FUNCTION_BLOCK "GCS7_M_Mixer"	// FB 54
TITLE = Mixer: Motor with 2 Digital Input
//  
//COPYRIGHT:    (C) 1997  BUHLER AG, CH-9240 UZWIL,  SWITZERLAND
//
//PRODUCT:      GCS7
//
//TITLE:        FB 54 MACHINE-CONTROL:Mixer:Motor with 2 Digital Input
//
//-------------------------------------------------------------------------
//
//IDENT:        AUTHOR:             DEPT:                       DATE:
//
//FB54.4.0      A. Egli             CT3                         17-Jun-2002
//              New Release with one block 
//FB54.3.1      A. Egli             CT3                         20-Mar-2000
//              Reset after mix done if mixer is open 
//FB54.3.0      A. Egli             CT3                         11-Oct-1999
//              Local data reduced 
//FB54.2B       K. Tischer          MU664                       06-Mar-1999
//              CC FC2 not UC FC2
//FB54.2A       A. Egli             CT3                         04-Mai-1998
//              StFault = StCode 32
//FB54.1A       A.Egli              AEE61                       5-Jul-1997
//              1st Release in S7
//
//-------------------------------------------------------------------------
//
//PURPOSE:      MANUAL : see [LL.MIXxxMAN]
//
//RESTRICTIONS: S7
//              ACCU2: Pointer to dynamic datas of the machine
//              ACCU1: Pointer to parameter datas of the machine
//
//-------------------------------------------------------------------------
//
AUTHOR : EA
FAMILY : GCS7LL
NAME : Mixer
VERSION : 4.0
VAR
  Ma : UDT 20540;
  Mon1 : FB 14;	//Element
  Mon2 : FB 14;	//Element
  Motor : FB 12;	//Element
END_VAR
VAR_TEMP
  tmpFaultStop : BOOL ;
  tmpFaultSum : BOOL ;
  tmpLocal : BOOL ;
  tmpLenDyn : INT ;
END_VAR
BEGIN
NETWORK
TITLE =
      L     22;
      T     #tmpLenDyn;
NETWORK
TITLE = PC Control
//=== Test Object number =====================
      L     "SYS_DirectCtrlDB".PC.ObjectNo;	//PCControl.ObjectNo
      L     #Ma.Par.ParObjectNo;	//Input ObjectNo
      <>I;
      JC    aEnd;
//=== Test OType      ========================
      L     2054;	//Input object type
      L     "SYS_DirectCtrlDB".PC.ObjectType;	//PCControl.ObjectType
      <>I;
      JC    aEnd;
//=== Test Handshake =========================
      A     "SYS_DirectCtrlDB".PC.Hsk.FExamine;	// Handshake.FExamine
      JC    aExa;
      A     "SYS_DirectCtrlDB".PC.Hsk.FDefineCmd;	// Handshake.FDefineCmd
      JC    aCmd;
      A     "SYS_DirectCtrlDB".PC.Hsk.FDefinePara;	// Handshake.FDefinePara
      JC    aPar;
aIni: L     2;	// FcInit
      UC    "SYS_DirectCtrl";
      JU    aEnd;
// Write parameter 
aPar: LAR1  P#DBX 58.0;
      L     P#6.0;
      +AR1;
      L     DBW [AR1,P#4.0];
      T     #Ma.Par.ParAfterMixTime;
// Write new commands from PC to Interface of group 
aCmd: A     "SYS_DirectCtrlDB".PC.Cmd1[8];	//Cmd1[8]=CmdOff
      S     #Ma.CmdOff;
      A     "SYS_DirectCtrlDB".PC.Cmd1[9];	//Cmd1[9]=CmdOn
      S     #Ma.CmdOn;
      A     "SYS_DirectCtrlDB".PC.Cmd1[10];	//Cmd1[10]=CmdNext
      S     #Ma.CmdNext;
      A     "SYS_DirectCtrlDB".PC.Cmd1[11];	//Cmd1[11]=CmdFaultReset
      S     #Ma.CmdFaultReset;
      A     "SYS_DirectCtrlDB".PC.Cmd1[13];	//Cmd1[13]=CmdManualOn
      S     #Ma.InManual;
      A     "SYS_DirectCtrlDB".PC.Cmd2[13];	//Cmd2[13]=CmdManualOff
      R     #Ma.InManual;
      A     "SYS_DirectCtrlDB".PC.Cmd1[6];	//Cmd1[14]=SlowOn
      S     #Motor.InOutManSlow;
      A     "SYS_DirectCtrlDB".PC.Cmd2[6];	//Cmd2[14]=SlowOff
      R     #Motor.InOutManSlow;
//Define Value
      AN    "SYS_DirectCtrlDB".PC.Hsk.FDefineValue;	// PC.Hsk.FDefineValue
      ON    #Ma.InManual;
      JC    aIni;
      LAR1  P#DBX 58.0;
      L     DBW [AR1,P#6.0];
      T     #Ma.InPreMixTime;
      L     DBW [AR1,P#8.0];
      T     #Ma.InMainMixTime;
      JU    aIni;
aExa: TAR2;	// Address Dynamic datas
      T     "SYS_DirectCtrlDB".GC.InDynAddr;	// -->PCControl.GC.InDynAddr
      L     #tmpLenDyn;	// Length Dynamic data
      T     "SYS_DirectCtrlDB".GC.InDynLen;	// -->PCControl.GC.InDynLen
      L     0;
      T     "SYS_DirectCtrlDB".GC.InParaAddr;	// -->PCControl.GC.InParaAddr
      T     "SYS_DirectCtrlDB".GC.InParaLen;	// -->PCControl.GC.InParaLen
      L     1;	// Code FcExamine
      UC    "SYS_DirectCtrl";
      L     10;	//Revision
      T     "SYS_DirectCtrlDB".GC.Revision;
aEnd: NOP   0;
NETWORK
TITLE = Interlocking
//===Global Group Orders===
      A     "GCS7_Gr_OutManualOn";	//Gr.OutManualOn
      S     #Ma.InManual;
      A     "GCS7_Gr_OutManualOff";	//Gr.OutManualOff
      R     #Ma.InManual;
      A     #Ma.InManual;
      S     "GCS7_Gr_InManual";	//Gr.InManual
      A     #Ma.InLocal;
      AN    #Ma.InManual;
      =     #tmpLocal;
//---Emptied
      A     #Ma.OutMainMixDone;
      A     #Ma.InOpen;
      S     #Ma.OutEmptied;
      AN    #Ma.OutMainMixDone;
      R     #Ma.OutEmptied;
//----New batch
      AN    #Ma.InRunPreMix;
      AN    #Ma.InRunMainMix;
      O     #Ma.CmdNewBatch;
      R     #Ma.OutEmptied;
      R     #Ma.OutPreMixIsOn;
      R     #Ma.OutPreMixDone;
//--- Fault----
      A     #Mon1.StFault;
      O     #Mon2.StFault;
      O     #Motor.StFault;
      =     #tmpFaultSum;
      =     #tmpFaultStop;
//--- Motor----
      AN    #Ma.OutAfterMixDone;
      O     #Ma.OutEmptied;
      O     #Ma.InManual;
      A     #Ma.InEnable;
      AN    #tmpFaultStop;
      A(;
      A     #Mon2.InpTrue;
      O     #Ma.Par.ParMon2IsLS;
      ON    #Ma.Par.ParWithMon2;
      );
      A(;
      A     #Mon1.InpTrue;
      ON    #Ma.Par.ParWithMon1;
      );
      AN    #Ma.CmdOff;
      =     #Motor.InEnableFwd;
      AN    #Ma.OutMainMixDone;
      O     #Ma.OutEmptied;
      A     #Ma.CmdNext;
      AN    #Ma.InManual;
      O;
      A     #Ma.InManual;
      A     #Ma.CmdOn;
      S     #Motor.CmdNext;
      A     #Ma.InSeqStop;
      AN    #Ma.InManual;
      =     #Motor.InSeqStop;
//--- Local mode --
      A     #tmpLocal;
      =     #Motor.InLocal;
      A     #Motor.StStopped;
      A     #tmpLocal;
      =     #Mon1.InLocal;
      =     #Mon2.InLocal;
//--- Monitoring
      SET;
      =     #Mon1.InMonTrue;
      A     #Motor.StStartedFwd;
      O     #Motor.StStartedRev;
      O     #Ma.Par.ParMon2IsLS;
      =     #Mon2.InMonTrue;
//--- Fault Reset -------------
      A     #Ma.CmdFaultReset;
      S     #Motor.CmdFaultReset;
      S     #Mon1.CmdFaultReset;
      S     #Mon2.CmdFaultReset;
NETWORK
TITLE = Mixing time
      L     0;
      L     #Ma.OutMixTime;
      >=I;
      JC    mix;
      AN    "GCS7_Gr_OutTick1s";	//Gr.OutTick1s
      ON    #Motor.StStartedFwd;
      JC    mix;
      +     -1;
      T     #Ma.OutMixTime;
//Pre mixing time 
mix:  AN    #Ma.InRunPreMix;
      AN    #Ma.InRunMainMix;
      R     #Ma.OutPreMixIsOn;
      R     #Ma.OutPreMixDone;
      JC    m2;
      A     #Ma.OutPreMixDone;
      JC    m2;
      A     #Ma.OutPreMixIsOn;
      JC    m12;
      S     #Ma.OutPreMixIsOn;
      L     #Ma.InPreMixTime;
      T     #Ma.OutMixTime;
m12:  L     #Ma.OutMixTime;
      L     0;
      <=I;
      R     #Ma.OutPreMixIsOn;
      S     #Ma.OutPreMixDone;
//Main mixing time 
m2:   AN    #Ma.InRunMainMix;
      ON    #Ma.OutPreMixDone;
      R     #Ma.OutMainMixIsOn;
      R     #Ma.OutMainMixDone;
      JC    m3;
      A     #Ma.OutMainMixDone;
      JC    m3;
      A     #Ma.OutMainMixIsOn;
      JC    m22;
      S     #Ma.OutMainMixIsOn;
      L     #Ma.InMainMixTime;
      T     #Ma.OutMixTime;
m22:  L     #Ma.OutMixTime;
      L     0;
      <=I;
      R     #Ma.OutMainMixIsOn;
      S     #Ma.OutMainMixDone;
//After mixing time 
m3:   AN    #Ma.OutMainMixDone;
      O     #Ma.InOpen;
      O     #Ma.OutEmptied;
      R     #Ma.OutAfterMixIsOn;
      R     #Ma.OutAfterMixDone;
      JC    m4;
      A     #Ma.OutAfterMixDone;
      JC    m4;
      A     #Ma.OutAfterMixIsOn;
      JC    m32;
      S     #Ma.OutAfterMixIsOn;
      L     #Ma.Par.ParAfterMixTime;
      T     #Ma.OutMixTime;
m32:  L     #Ma.OutMixTime;
      L     0;
      <=I;
      R     #Ma.OutAfterMixIsOn;
      S     #Ma.OutAfterMixDone;
NETWORK
TITLE = Call Digital Input: Monitor B1
m4:   AN    #Ma.Par.ParWithMon1;
      JC    m5;
      CALL  #Mon1;
NETWORK
TITLE = Call Digital Input: Monitor B2
m5:   AN    #Ma.Par.ParWithMon2;
      JC    Moto;
      CALL  #Mon2;
NETWORK
TITLE = Call Motor
Moto: CALL  #Motor;
NETWORK
TITLE = Jump to actual state
      A     #Ma.StStopped;
      JC    S0;	// ===> State
      A     #Ma.StStarted;
      JC    S2;	// ===> State
      A     #Ma.StStarting;
      JC    S1;	// ===> State
      A     #Ma.StStopping;
      JC    S3;	// ===> State
      A     #Ma.StFault;
      JC    S4;	// ===> State
NETWORK
TITLE = Stopped
xxS0: S     #Ma.StStopped;
S0:   A     #tmpFaultSum;
      R     #Ma.StStopped;
      JC    xxS4;	//--> StFault
      AN    #Motor.StStopped;
      R     #Ma.StStopped;
      JC    xxS1;	//--> StStarting
      JU    OUT;
NETWORK
TITLE = Starting
xxS1: S     #Ma.StStarting;
S1:   A     #tmpFaultSum;
      R     #Ma.StStarting;
      JC    xxS4;	//--> StFault
// Condition for StStopping
      A     #Motor.StStopped;
      O     #Motor.StStopping;
      R     #Ma.StStarting;
      JC    xxS3;	//--> StStopping
      AN    #Mon1.StTrue;
      A     #Ma.Par.ParWithMon1;
      O;
      AN    #Mon2.StTrue;
      A     #Ma.Par.ParWithMon2;
      JC    S2En;
// Condition for StStartedFwd
      A     #Motor.StStartedFwd;
      R     #Ma.StStarting;
      JC    xxS2;	//--> StStartedFwd
S2En: JU    OUT;
NETWORK
TITLE = StartedFwd
xxS2: S     #Ma.StStarted;
S2:   A     #tmpFaultSum;
      R     #Ma.StStarted;
      JC    xxS4;	//--> StFault
// Condition for StStopping
      AN    #Motor.StStartedFwd;
      R     #Ma.StStarted;
      JC    xxS3;	//--> StStopping
      JU    OUT;
NETWORK
TITLE = Stopping
xxS3: S     #Ma.StStopping;
S3:   A     #tmpFaultSum;
      R     #Ma.StStopping;
      JC    xxS4;	//--> StFault
// Condition for StStopped
      A     #Motor.StStopped;
      R     #Ma.StStopping;
      JC    xxS0;	//--> StStopped
// Condition for StStarting
      AN    #Motor.StStopping;
      R     #Ma.StStopping;
      JC    xxS1;	//--> StStarting
      JU    OUT;
NETWORK
TITLE = Fault
xxS4: S     #Ma.StFault;
S4:   AN    #tmpFaultSum;
      R     #Ma.StFault;
      JC    xxS3;	//--> StStopping
      JU    OUT;
NETWORK
TITLE = Global End
OUT:  CLR;	//---Clear all commands
      =     #Ma.CmdOn;
      =     #Ma.CmdOff;
      =     #Ma.CmdNext;
      =     #Ma.CmdFaultReset;
      =     #Ma.CmdNewBatch;
NETWORK
TITLE = State Code
// Same as motor
      L     32;	// StCode=Fault
      A     #Ma.StFault;
      JC    Code;
//Started
      AN    #Ma.StStarted;
      JC    C2;
      A     #Ma.OutPreMixIsOn;
      AN    #Ma.OutEmptied;
      L     4;	// StCode=Premix
      JC    Code;
      A     #Ma.OutMainMixIsOn;
      AN    #Ma.OutEmptied;
      L     5;	// StCode=MainMix
      JC    Code;
      A     #Ma.OutAfterMixIsOn;
      AN    #Ma.OutEmptied;
      L     6;	// StCode=AfterMix
      JC    Code;
      L     3;	// StCode=Started
      JU    Code;
//Stopped
C2:   AN    #Ma.StStopped;
      JC    C1;
      A     #Ma.OutMainMixDone;
      AN    #Ma.OutEmptied;
      L     8;	// StCode=Wait
      JC    Code;
      L     1;	// StCode=Stopped
      JU    Code;
//Starting
C1:   A     #Ma.StStarting;
      L     2;	// StCode=Starting
      JC    Code;
//Stopping
      L     7;	// StCode=Stopping
Code: L     #Ma.StCode;	// Old state code
      TAK;
      T     #Ma.StCode;	// Save state code
      <>I;
      L     3;
      CC    "SYS_CBitCtrl";	//Set change bit
END_FUNCTION_BLOCK

FUNCTION_BLOCK "GCS7_M_DFZK"	// FB 55
TITLE = DFZK vertical rotor mill
//  
//COPYRIGHT:    (C) 2000  BUHLER AG, CH-9240 UZWIL, SWITZERLAND
//
//PRODUCT:      GCS7
//
//TITLE:        FB55 Machine Control: DFZK vertical rotor mill
//
//-------------------------------------------------------------------------
//
//IDENT:        AUTHOR:             DEPT:                       DATE:
//
//FB55.2.3      A.Egli              CT3                         21.1.2005
//              For Screen change check input button
//FB55.2.2      A.Egli              FU53                        18.05.2004
//              Reset Manual mode when mill is not in automatic
//FB55.2.1      A.Egli              FU53                        15.03.2004
//              DFCM Freigabe koordinieren
//              Transition to StStopping if only one of both mill used
//              (Change [1.6] and [1.6a] from B.Thoma 
//FB55.2.0      A. Egli             CT3                         17-Jun-2002
//              New Release with one block 
//FB55.1.5      A.Egli              CT3                         14.09.2001
//              Condition B201LS.InMonTrue,B250LS.InMonTrue
//FB55.1.4      A.Egli              CT3                         14.09.2001
//              Unlock Cone in StNoPosition 
//FB55.1.3      B.Thoma             FU53                        21.01.2001
//              Monitoring Metal purifying if ma.ststarted 
//FB55.1.2      S. Kalberer         CT3                         21.11.2000
//              Avoid simultaneous brake event with global flag M 12.0
//FB55.1.1      S. Kalberer         CT3                         02.10.2000
//              Process of elements B201LS + 250LS (clam-gates) adapted
//FB55.1.0      S. Kalberer         CT3                         06.06.2000
//              1st Release in S7
//FB55.0.3      S. Kalberer         CT3                         26.05.2000
//              Cone open/close adapted
//FB55.0.2      S. Kalberer         CT3                         03.05.2000
//              Empty run without DFCM
//FB55.0.1      S. Kalberer         CT3                         26.04.2000
//              Segment gate parameter changed
//FB55.0.0      S. Kalberer         CT3                         20.04.2000
//              Software brake event and speed change
//
//-------------------------------------------------------------------------
//
//PURPOSE:      MANUAL : see [LL.VRMillENMAN]
//
//RESTRICTIONS: S7
//              ACCU2: Pointer to dynamic datas of the machine
//              ACCU1: Pointer to parameter datas of the machine
//
//-------------------------------------------------------------------------
//
AUTHOR : EA
FAMILY : GCS7LL
NAME : DFZKVRMi
VERSION : 2.3
VAR
  Ma : UDT 20550;
  M200 : FB 12;	//Element
  M300 : FB 12;	//Element
  M350 : FB 12;	//Element
  DFCMMill1 : FB 12;	//Element
  DFCMMill2 : FB 12;	//Element
  Y203V : FB 13;	//Element
  Y302V_Y305V : FB 13;	//Element
  Y352V_Y355V : FB 13;	//Element
  Y307V_Y309V : FB 13;	//Element
  Y357V_Y359V : FB 13;	//Element
  A316VI : FB 14;	//Element
  A366VI : FB 14;	//Element
  B205LS : FB 14;	//Element
  B206HL : FB 14;	//Element
  B201LS : FB 14;	//Element
  B250LS : FB 14;	//Element
  B300SM : FB 14;	//Element
  B350SM : FB 14;	//Element
  B310LS : FB 14;	//Element
  B360LS : FB 14;	//Element
  B317HL : FB 14;	//Element
  B367HL : FB 14;	//Element
  A209LC_AO1 : FB 17;	//Element
  A209LC_AO2 : FB 17;	//Element
  A209LC_AI1 : FB 19;	//Element
  A209LC_AI2 : FB 19;	//Element
  Y251V_52_53_54V : FB 20;	//Element
END_VAR
VAR_TEMP
  tmpFaultSum : BOOL ;	// Summary faults
  tmpFaultStopFeedingMill1 : BOOL ;	// Relevant faults to stop feeding mill 1
  tmpFaultStopFeedingMill2 : BOOL ;	// Relevant faults to stop feeding mill 2
  tmpFaultImmStopMill1 : BOOL ;	// Relevant faults to stop mill 1 immediately
  tmpFaultImmStopMill2 : BOOL ;	// Relevant faults to stop mill 2 immediately
  tmpFaultStopAfEmptyMill1 : BOOL ;	// Relevant faults to stop mill 2 after emptying time
  tmpFaultStopAfEmptyMill2 : BOOL ;	// Relevant faults to stop mill 1 after emptying time
  tmpEnableMill1 : BOOL ;
  tmpEnableMill2 : BOOL ;	//[1.2] ParMa.OutScreenChMill1 = tmpOutScreenChangeMill1 : BOOL; // Signal screen
  tmpSpeedChangeMill1 : BOOL ;	// Speed change requested mill 1
  tmpSpeedChangeMill2 : BOOL ;	// Speed change requested mill 1
  tmpTriggerFlag : BOOL ;
  tmpLenDyn : INT ;
END_VAR
BEGIN
NETWORK
TITLE =
      L     106;
      T     #tmpLenDyn;
NETWORK
TITLE = PC Control
//=== Test Object number =====================
      L     "SYS_DirectCtrlDB".PC.ObjectNo;	//PCControl.ObjectNo
      L     #Ma.Par.ParObjectNo;	//Input ObjectNo
      <>I;
      JC    aEnd;
//=== Test OType  ========================
      L     2055;	//Input object type
      L     "SYS_DirectCtrlDB".PC.ObjectType;	//PCControl.ObjectType
      <>I;
      JC    aEnd;
//=== Test Handshake =========================
      A     "SYS_DirectCtrlDB".PC.Hsk.FExamine;	// Handshake.FExamine
      JC    aExa;
      A     "SYS_DirectCtrlDB".PC.Hsk.FDefineCmd;	// Handshake.FDefineCmd
      JC    aCmd;
      A     "SYS_DirectCtrlDB".PC.Hsk.FDefinePara;	// Handshake.FDefinePara
      JC    pPar;
aIni: L     2;	// FcInit
      UC    "SYS_DirectCtrl";
      JU    aEnd;
// Write parameter 
pPar: LAR1  P#DBX 58.0;
      L     P#6.0;
      +AR1;
      L     DBW [AR1,P#4.0];
      L     "SYS_DirectCtrlDB".PC.Value[25];	//PCControl.PC.Value[25]
      T     #Ma.Par.ParEmptyRunMill1;
      L     "SYS_DirectCtrlDB".PC.Value[26];	//PCControl.PC.Value[26]
      T     #Ma.Par.ParEmptyRunMill2;
      L     "SYS_DirectCtrlDB".PC.Value[27];	//PCControl.PC.Value[27]
      T     #Ma.Par.ParEmptyTimeMill1;
      L     "SYS_DirectCtrlDB".PC.Value[28];	//PCControl.PC.Value[28]
      T     #Ma.Par.ParEmptyTimeMill2;
      L     "SYS_DirectCtrlDB".PC.Value[29];	//PCControl.PC.Value[29]
      T     #Ma.Par.ParBrakeTimeMill1;
      L     "SYS_DirectCtrlDB".PC.Value[30];	//PCControl.PC.Value[30]
      T     #Ma.Par.ParBrakeTimeMill2;
      L     "SYS_DirectCtrlDB".PC.Value[31];	//PCControl.PC.Value[31]
      T     #Ma.Par.ParSwitchChTime;
// Write new commands from PC to Interface of group 
aCmd: A     "SYS_DirectCtrlDB".PC.Cmd1[0];	//Cmd1[0]=CmdBrakeMill1On
      S     #Ma.InBrakeMill1;
      A     "SYS_DirectCtrlDB".PC.Cmd2[0];	//Cmd2[0]=CmdBrakeMill1Off
      R     #Ma.InBrakeMill1;
      A     "SYS_DirectCtrlDB".PC.Cmd1[1];	//Cmd1[1]=CmdBrakeMill2On
      S     #Ma.InBrakeMill2;
      A     "SYS_DirectCtrlDB".PC.Cmd2[1];	//Cmd2[1]=CmdBrakeMill2Off
      R     #Ma.InBrakeMill2;
      A     "SYS_DirectCtrlDB".PC.Cmd1[6];	//Cmd1[6]=CmdUsedMill1On
      S     #Ma.InUsedMill1;
      A     "SYS_DirectCtrlDB".PC.Cmd2[6];	//Cmd2[6]=CmdUsedMill1Off
      R     #Ma.InUsedMill1;
      A     "SYS_DirectCtrlDB".PC.Cmd1[7];	//Cmd1[7]=CmdUsedMill2On
      S     #Ma.InUsedMill2;
      A     "SYS_DirectCtrlDB".PC.Cmd2[7];	//Cmd2[7]=CmdUsedMill2Off
      R     #Ma.InUsedMill2;
      A     "SYS_DirectCtrlDB".PC.Cmd1[10];	//Cmd1[10]=CmdNext
      S     #Ma.CmdNext;
      A     "SYS_DirectCtrlDB".PC.Cmd1[11];	//Cmd1[11]=CmdFaultReset
      S     #Ma.CmdFaultReset;
      JU    aIni;
aExa: TAR2;	// Address Dynamic datas
      T     "SYS_DirectCtrlDB".GC.InDynAddr;	// -->PCControl.GC.InDynAddr
      L     #tmpLenDyn;	// Length Dynamic data
      T     "SYS_DirectCtrlDB".GC.InDynLen;	// -->PCControl.GC.InDynLen
      L     0;
      T     "SYS_DirectCtrlDB".GC.InParaAddr;	// -->PCControl.GC.InParaAddr
      T     "SYS_DirectCtrlDB".GC.InParaLen;	// -->PCControl.GC.InParaLen
      L     1;	// Code FcExamine
      UC    "SYS_DirectCtrl";
      L     10;	//Revision
      T     "SYS_DirectCtrlDB".GC.Revision;
aEnd: NOP   0;
NETWORK
TITLE = General conditions
      NOP   0;
//=== Condition to set hardware brake output
// Mill1
      A     #Ma.OutBrakeMill1;	// No brake condition
      AN    #Ma.OutLoadedMill1;	// Mill 1 is loaded with product
      AN    #Ma.Par.OutSpeedChMill1;	// Mill 1 is speed changing
      AN    #Ma.OutFastMill1;
      AN    #Ma.Par.OutBrakeAcvMill1;	// Brake event is active
      AN    #Ma.OutpBrakeMill2;	// Mill 2 is braking
      S     #Ma.OutpBrakeMill1;
// Mill2
      A     #Ma.OutBrakeMill2;	// No brake condition
      AN    #Ma.OutLoadedMill2;	// Mill 2 is loaded with product
      AN    #Ma.Par.OutSpeedChMill2;	// Mill 2 is speed changing
      AN    #Ma.OutFastMill2;
      AN    #Ma.Par.OutBrakeAcvMill2;	// Brake event is active
      AN    #Ma.OutpBrakeMill1;	// Mill 1 is braking
      S     #Ma.OutpBrakeMill2;
//=== Speed change
      A(;	// Condition to change speed mill 1
      AN    #Ma.InFastMill;
      A     #Ma.OutFastMill1;
      O;
      A     #Ma.OutFastMill1;
      A     #Ma.OutBrakeMill1;
      O;
      A     #Ma.InFastMill;
      AN    #Ma.OutFastMill1;
      AN    #Ma.OutBrakeMill1;
      );
      AN    #M300.StStopped;
      AN    #M300.StFault;
      A     #M300.Par.Par2Speed;
      =     #tmpSpeedChangeMill1;
      S     #Ma.Par.OutSpeedChMill1;	// Indicate speed changing mill 1
      A     #M300.StStartedFwd;	//--- If motor is started again 
      O     #M300.StStartedRev;
      AN    #tmpSpeedChangeMill1;
      O     #M300.StFault;	// or fault
      R     #Ma.Par.OutSpeedChMill1;	// --> Speed changing is done mill 1
//        
      A(;	// Condition to change speed mill 2
      AN    #Ma.InFastMill;
      A     #Ma.OutFastMill2;
      O;
      A     #Ma.OutFastMill2;
      A     #Ma.OutBrakeMill2;
      O;
      A     #Ma.InFastMill;
      AN    #Ma.OutFastMill2;
      AN    #Ma.OutBrakeMill2;
      );
      AN    #M350.StStopped;
      AN    #M350.StFault;
      A     #M350.Par.Par2Speed;
      =     #tmpSpeedChangeMill2;
      S     #Ma.Par.OutSpeedChMill2;	// Indicate speed changing mill 2
      A     #M350.StStartedFwd;	//--- If motor is started again 
      O     #M350.StStartedRev;
      AN    #tmpSpeedChangeMill2;
      O     #M350.StFault;	// or fault
      R     #Ma.Par.OutSpeedChMill2;	// --> Speed changing is done mill 2
NETWORK
TITLE = Prepare brake mills
// Programming the following functions:
// - Brake the motor (changing the direction) by request screen change
//   or InBrake signal
// - Stop only one mill at once
      NOP   0;
//=== Prepare brake mill 1
// Request screen change
      L     #Ma.InScreenNoMill1;	// Check for new screen number
      L     #Ma.OutScreenNoAcMill1;
      <>I;
      A     #Ma.InUsedMill1;
      AN    "GCS7_Gr_InBrakeMill";	//[1.2->] Gr.InBrakeMill
      S     #Ma.Par.OutScreenChMill1;	// Screen change mill 1
      L     #Ma.InScreenNoMill1;	// Check for new screen number
      L     #Ma.OutScreenNoAcMill1;
      ==I;
      ON    #Ma.InUsedMill1;
      R     #Ma.Par.OutScreenChMill1;	//[<-1.2] Screen change mill 1
      A     #Ma.Par.OutScreenChMill1;	// Screennumber different to acutal screen
      O     #Ma.Par.OutBrakeAcvMill1;	// or brake signal
      O     #Ma.InBrakeMill1;
      AN    #M300.StStopped;
      AN    #M300.StStopping;
      AN    #M300.StFault;
      AN    #M300.StStarting;
      AN    "GCS7_Gr_InBrakeMill";	//[1.2] Gr.InBrakeMill
      S     "GCS7_Gr_InBrakeMill";	//[1.2] Gr.InBrakeMill
      S     #Ma.OutBrakeMill1;
//=== Prepare brake mill 2
// Request screen change
      L     #Ma.InScreenNoMill2;	// Check for new screen number
      L     #Ma.OutScreenNoAcMill2;
      <>I;
      A     #Ma.InUsedMill2;
      A     #Ma.Par.ParWithMill2;
      AN    "GCS7_Gr_InBrakeMill";	//[1.2->] Gr.InBrakeMill
      S     #Ma.Par.OutScreenChMill2;	// Screen change mill 2
      L     #Ma.InScreenNoMill2;	// Check for new screen number
      L     #Ma.OutScreenNoAcMill2;
      ==I;
      ON    #Ma.InUsedMill2;
      ON    #Ma.Par.ParWithMill2;
      R     #Ma.Par.OutScreenChMill2;	//[<-1.2] Screen change mill 2
      A     #Ma.Par.ParWithMill2;
      JCN   PBrE;
      A     #Ma.Par.OutScreenChMill2;	// Screennumber different to acutal screen
      O     #Ma.Par.OutBrakeAcvMill2;	// or brake signal
      O     #Ma.InBrakeMill2;
      AN    #M350.StStopped;
      AN    #M350.StStopping;
      AN    #M350.StFault;
      AN    #M350.StStarting;
      AN    "GCS7_Gr_InBrakeMill";	//[1.2] Gr.InBrakeMill
      S     "GCS7_Gr_InBrakeMill";	//[1.2] Gr.InBrakeMill
      S     #Ma.OutBrakeMill2;
PBrE: NOP   0;
NETWORK
TITLE = Handle emptying timer
// OutLoadedMillX will be set if once product was feeded (OutFeedingMillX were 
//set once).
      A     #Ma.OutLoadedMill1;	//=== Condition for emptying mill 1
      A(;
      ON    #Ma.OutFeedingMill1;
      O     #Ma.OutBrakeMill1;
      O     #Ma.InAlarmTempMill1;
      O     #Ma.InAlarmTempMill2;
      );
      JC    Em11;
      R     #Ma.OutEmptyingMill1;
      L     0;
      T     #Ma.OutEmptyTimeMill1;
      JU    Em20;
Em11: A     #Ma.OutEmptyingMill1;	// Emptying time is active
      JC    Em12;
      S     #Ma.OutEmptyingMill1;
      L     #Ma.Par.ParEmptyTimeMill1;	// Set emptying time
      T     #Ma.OutEmptyTimeMill1;
Em12: AN    "GCS7_Gr_OutTick500ms";	// Gr.OutTick500ms (M 10.4)
      L     #Ma.OutEmptyTimeMill1;
      JC    Em13;
      +     -5;	// Decrement timer
      T     #Ma.OutEmptyTimeMill1;
Em13: L     0;
      <=I;
      R     #Ma.OutLoadedMill1;
      R     #Ma.OutEmptyingMill1;
      S     #Ma.OutEmptyingDoneMill1;
Em20: A     #Ma.OutLoadedMill2;	//=== Condition for emptying mill 2
      A(;
      ON    #Ma.OutFeedingMill2;
      O     #Ma.OutBrakeMill2;
      O     #Ma.InAlarmTempMill1;
      O     #Ma.InAlarmTempMill2;
      );
      JC    Em21;
      R     #Ma.OutEmptyingMill2;
      L     0;
      T     #Ma.OutEmptyTimeMill2;
      JU    Em30;
Em21: A     #Ma.OutEmptyingMill2;	// Emptying time is active
      JC    Em22;
      S     #Ma.OutEmptyingMill2;
      L     #Ma.Par.ParEmptyTimeMill2;	// Set emptying time
      T     #Ma.OutEmptyTimeMill2;
Em22: AN    "GCS7_Gr_OutTick500ms";	// Gr.OutTick500ms (M 10.4)
      L     #Ma.OutEmptyTimeMill2;
      JC    Em23;
      +     -5;	// Decrement timer
      T     #Ma.OutEmptyTimeMill2;
Em23: L     0;
      <=I;
      R     #Ma.OutLoadedMill2;
      R     #Ma.OutEmptyingMill2;
      S     #Ma.OutEmptyingDoneMill2;
Em30: NOP   0;
NETWORK
TITLE = Handle switch change timer
      NOP   0;
//=== Condition for switch change time mill 1
      A     #M300.StStartedFwd;
      O     #M300.StStartedRev;
      A(;
      A     #Ma.OutBrakeMill1;	// Run time before brake
      AN    #Ma.Par.OutBrakeAcvMill1;
      AN    #Ma.Par.OutSpeedChMill1;
      O     #tmpSpeedChangeMill1;	// Run time at speed change
      );
      O     #Ma.Par.OutSwitchChMill1;
      AN    #Ma.OutEmptyingMill1;
      AN    #Ma.OutFeedingMill1;
      JC    Ch11;
      R     #Ma.Par.OutSwitchChMill1;
      L     0;
      T     #Ma.OutSwitchChTimeMill1;
      JU    Ch20;
Ch11: A     #Ma.Par.OutSwitchChMill1;	// Change time is active
      JC    Ch12;
      S     #Ma.Par.OutSwitchChMill1;
      L     #Ma.Par.ParSwitchChTime;	// Set switch change time
      T     #Ma.OutSwitchChTimeMill1;
Ch12: AN    "GCS7_Gr_OutTick500ms";	// Gr.OutTick500ms (M 10.4)
      L     #Ma.OutSwitchChTimeMill1;
      JC    Ch13;
      +     -5;	// Decrement timer
      T     #Ma.OutSwitchChTimeMill1;
Ch13: L     0;
      <=I;
      R     #Ma.Par.OutSwitchChMill1;
      S     #Ma.Par.OutSwitchChDoneMill1;
//=== Condition for switch change time mill 2
Ch20: A     #M350.StStartedFwd;
      O     #M350.StStartedRev;
      A(;
      A     #Ma.OutBrakeMill2;	// Run time before brake
      AN    #Ma.Par.OutBrakeAcvMill2;
      AN    #Ma.Par.OutSpeedChMill2;
      O     #tmpSpeedChangeMill2;	// Run time at speed change
      );
      O     #Ma.Par.OutSwitchChMill2;
      AN    #Ma.OutEmptyingMill2;
      AN    #Ma.OutFeedingMill2;
      JC    Ch21;
      R     #Ma.Par.OutSwitchChMill2;
      L     0;
      T     #Ma.OutSwitchChTimeMill2;
      JU    Ch30;
Ch21: A     #Ma.Par.OutSwitchChMill2;	// Change time is active
      JC    Ch22;
      S     #Ma.Par.OutSwitchChMill2;
      L     #Ma.Par.ParSwitchChTime;	// Set switch change time
      T     #Ma.OutSwitchChTimeMill2;
Ch22: AN    "GCS7_Gr_OutTick500ms";	// Gr.OutTick500ms (M 10.4)
      L     #Ma.OutSwitchChTimeMill2;
      JC    Ch23;
      +     -5;	// Decrement timer
      T     #Ma.OutSwitchChTimeMill2;
Ch23: L     0;
      <=I;
      R     #Ma.Par.OutSwitchChMill2;
      S     #Ma.Par.OutSwitchChDoneMill2;
Ch30: NOP   0;
NETWORK
TITLE = Handle brake timer
// Programming the following functions:
// - Brake the motors
      A     #Ma.OutpBrakeMill1;	//=== Brake mill 1
      AN    #Ma.Par.OutSwitchChMill1;
      JCN   Br20;
      A     #Ma.Par.OutBrakeAcvMill1;
      JC    Br11;
      S     #Ma.Par.OutBrakeAcvMill1;
      L     #Ma.Par.ParBrakeTimeMill1;	// Brake time mill 1
      T     #Ma.OutBrakeTimeMill1;
Br11: AN    #Ma.CmdTick100ms;
      L     #Ma.OutBrakeTimeMill1;
      JC    Br12;
      +     -1;	// Decrement timer
      T     #Ma.OutBrakeTimeMill1;
Br12: L     0;
      <=I;
      R     #Ma.OutpBrakeMill1;	// Brake mill 1
      R     "GCS7_Gr_InBrakeMill";	//[1.2] Gr.InBrakeMill
Br20: A     #Ma.OutpBrakeMill2;	//=== Brake mill 2
      AN    #Ma.Par.OutSwitchChMill2;
      JCN   Br30;
      A     #Ma.Par.OutBrakeAcvMill2;
      JC    Br21;
      S     #Ma.Par.OutBrakeAcvMill2;
      L     #Ma.Par.ParBrakeTimeMill2;	// Brake time mill 2
      T     #Ma.OutBrakeTimeMill2;
Br21: AN    #Ma.CmdTick100ms;
      L     #Ma.OutBrakeTimeMill2;
      JC    Br22;
      +     -1;	// Decrement timer
      T     #Ma.OutBrakeTimeMill2;
Br22: L     0;
      <=I;
      R     #Ma.OutpBrakeMill2;	// Brake mill 2
      R     "GCS7_Gr_InBrakeMill";	//[1.2] Gr.InBrakeMill
Br30: NOP   0;
NETWORK
TITLE = Change screen / clear brake event
      NOP   0;
//Quit screen change mill 1 / clear InBrake event
      A     #Ma.InpS311Z6;	//--- Push button screen change acknowledge mill 1
      A     #Y307V_Y309V.StLN;	// Cone locked mill 1
      A     #Ma.Par.OutScreenChMill1;
      A     #Ma.Par.OutConeOpenedMill1;	// Was cone mill 1 opened?
      O;
      AN    #Ma.Par.OutScreenChMill1;	//--- Clear InBrake event
      AN    #Ma.OutpBrakeMill1;	// Mill is still braking
      AN    #Ma.InBrakeMill1;
      A     #B300SM.StTrue;	// Standstill mill 1
      JCN   Cs01;
      AN    #Ma.InpS311Z6;	//--- Push button screen change acknowledge mill 1 //[2.3]
      ON    #Ma.Par.OutScreenChMill1;	//[2.3]
      JC    SC1A;	//[2.3]
      L     #Ma.InScreenNoMill1;	// Set actual screen number
      T     #Ma.OutScreenNoAcMill1;
SC1A: R     #Ma.Par.OutConeOpenedMill1;
      R     #Ma.OutBrakeMill1;	// Clear brake event signal
      R     #Ma.Par.OutBrakeAcvMill1;
//Quit screen change mill 2 / clear InBrake event
Cs01: A     #Ma.InpS361Z6;	//--- Push button screen change acknowledge mill 2
      A     #Y357V_Y359V.StLN;	// Cone locked mill 2
      A     #Ma.Par.OutScreenChMill2;
      A     #Ma.Par.OutConeOpenedMill2;	// Was cone mill 2 opened?
      O;
      AN    #Ma.Par.OutScreenChMill2;	//--- Clear InBrake event
      AN    #Ma.OutpBrakeMill2;	// Mill is still braking
      AN    #Ma.InBrakeMill2;
      A     #B350SM.StTrue;	// Standstill mill 2
      ON    #Ma.Par.ParWithMill2;
      JCN   Cs02;
      AN    #Ma.InpS361Z6;	//--- Push button screen change acknowledge mill //[2.3]
      ON    #Ma.Par.OutScreenChMill2;	//[2.3]
      JC    SC2A;	//[2.3]
      L     #Ma.InScreenNoMill2;	// Set actual screen number
      T     #Ma.OutScreenNoAcMill2;
SC2A: R     #Ma.Par.OutConeOpenedMill2;
      R     #Ma.OutBrakeMill2;	// Clear brake event signal
      R     #Ma.Par.OutBrakeAcvMill2;
//Set signals: cones of mills 1 and 2 were opened
Cs02: AN    #Y302V_Y305V.StLN;	// Cone not closed mill 1
      A     #Y307V_Y309V.StHN;	// Cone locked mill 1
      A     #Ma.Par.OutScreenChMill1;
      S     #Ma.Par.OutConeOpenedMill1;
      AN    #Y352V_Y355V.StLN;	// Cone not closed mill 2
      A     #Y357V_Y359V.StHN;	// Cone locked mill 2
      A     #Ma.Par.OutScreenChMill2;
      S     #Ma.Par.OutConeOpenedMill2;
//Lamp request for screen change mill 1
      A     #Ma.Par.OutScreenChMill1;
      A     "SYS_Pulse500ms";	// All.Pulse500ms (M 9.3): f= 1 Hz
      =     #Ma.OutpS311Z6;	// Lamp request for screen change mill 1
//Lamp request for screen change mill 2
      A     #Ma.Par.OutScreenChMill2;
      A     "SYS_Pulse500ms";	// All.Pulse500ms (M 9.3): f= 1 Hz
      =     #Ma.OutpS361Z6;	// Lamp request for screen change mill 2
NETWORK
TITLE = Interlocking
      NOP   0;
//--- Summary fault----
      A     #M200.StFault;	// Fan DFAV
      O     #M300.StFault;	// Motor mill 1
      O     #M350.StFault;	// Motor mill 2
      O     #DFCMMill1.StFault;	// DFCM control unit mill 1
      O     #DFCMMill2.StFault;	// DFCM control unit mill 2
      O     #Y203V.StFault;	// Open dense-medium valve
      O     #Y302V_Y305V.StFault;	// Cone open/close mill 1
      O     #Y352V_Y355V.StFault;	// Cone open/close mill 2
      O     #Y307V_Y309V.StFault;	// Cone unlock/lock mill 1
      O     #Y357V_Y359V.StFault;	// Cone unlock/lock mill 2
      O     #A316VI.StFault;	// Vibration control mill 1
      O     #A366VI.StFault;	// Vibration control mill 2
      O     #B205LS.StFault;	// Metal purifying valve closed
      O     #B206HL.StFault;	// HL DFAV full
      O     #B201LS.StFault;	// Clam-gate mill 1 closed
      O     #B250LS.StFault;	// Clam-gate mill 2 closed
      O     #B300SM.StFault;	// Standstill mill 1
      O     #B350SM.StFault;	// Standstill mill 2
      O     #B310LS.StFault;	// Switch panel ok mill 1
      O     #B360LS.StFault;	// Switch panel ok mill 2
      O     #B317HL.StFault;	// HL cone mill 1 (backup)
      O     #B367HL.StFault;	// HL cone mill 2 (backup)
      O     #Y251V_52_53_54V.StFault;	// Flap box
      O     #Ma.InAlarmTempMill1;
      O     #Ma.InAlarmTempMill2;
      AN    #Ma.InLocal;
      =     #tmpFaultSum;
//--- Fault stop after emptying mill 1----
      O     #Ma.InAlarmTempMill1;
      O     #Ma.InAlarmTempMill2;
      AN    #Ma.InLocal;
      =     #tmpFaultStopAfEmptyMill1;
//--- Fault stop after emptying mill 2----
      O     #Ma.InAlarmTempMill1;
      O     #Ma.InAlarmTempMill2;
      AN    #Ma.InLocal;
      =     #tmpFaultStopAfEmptyMill2;
//--- Fault immediate stop mill 1----
      A     #M300.StFault;	// Motor mill 1
      O     #Y302V_Y305V.StFault;	// Cone open/close mill 1
      O     #Y352V_Y355V.StFault;	// Cone open/close mill 2
      O     #Y307V_Y309V.StFault;	// Cone unlock/lock mill 1
      O     #Y357V_Y359V.StFault;	// Cone unlock/lock mill 2
      O     #A316VI.StFault;	// Vibration control mill 1
      O     #B300SM.StFault;	// Standstill mill 1
      AN    #Ma.InLocal;
      =     #tmpFaultImmStopMill1;
//--- Fault immediate stop mill 2----
      O     #M350.StFault;	// Motor mill 2
      O     #Y302V_Y305V.StFault;	// Cone open/close mill 1
      O     #Y352V_Y355V.StFault;	// Cone open/close mill 2
      O     #Y307V_Y309V.StFault;	// Cone unlock/lock mill 1
      O     #Y357V_Y359V.StFault;	// Cone unlock/lock mill 2
      O     #A366VI.StFault;	// Vibration control mill 2
      O     #B350SM.StFault;	// Standstill mill 2
      AN    #Ma.InLocal;
      =     #tmpFaultImmStopMill2;
//--- Fault stop feeding mill 1----
      A     #M200.StFault;	// Fan DFAV
      O     #M300.StFault;	// Motor mill 1
      O     #M350.StFault;	// Motor mill 2
      O     #DFCMMill1.StFault;	// DFCM control unit mill 1
      O     #Y203V.StFault;	// Open dense-medium valve
      O     #Y302V_Y305V.StFault;	// Cone open/close mill 1
      O     #Y352V_Y355V.StFault;	// Cone open/close mill 2
      O     #Y307V_Y309V.StFault;	// Cone unlock/lock mill 1
      O     #Y357V_Y359V.StFault;	// Cone unlock/lock mill 2
      O     #A316VI.StFault;	// Vibration control mill 1
      O     #A366VI.StFault;	// Vibration control mill 2
      O     #B205LS.StFault;	// Metal purifying valve closed
      O     #B206HL.StFault;	// HL DFAV full
      O     #B300SM.StFault;	// Standstill mill 1
      O     #B350SM.StFault;	// Standstill mill 2
      O     #B317HL.StFault;	// HL cone mill 1 (backup)
      O     #B367HL.StFault;	// HL cone mill 2 (backup)
      O     #Y251V_52_53_54V.StFault;	// Flap box
      O     #Ma.InAlarmTempMill1;
      O     #Ma.InAlarmTempMill2;
      AN    #Ma.InLocal;
      =     #tmpFaultStopFeedingMill1;
//--- Fault stop feeding mill 2----
      A     #M200.StFault;	// Fan DFAV
      O     #M300.StFault;	// Motor mill 1
      O     #M350.StFault;	// Motor mill 2
      O     #DFCMMill2.StFault;	// DFCM control unit mill 2
      O     #Y203V.StFault;	// Open dense-medium valve
      O     #Y302V_Y305V.StFault;	// Cone open/close mill 1
      O     #Y352V_Y355V.StFault;	// Cone open/close mill 2
      O     #Y307V_Y309V.StFault;	// Cone unlock/lock mill 1
      O     #Y357V_Y359V.StFault;	// Cone unlock/lock mill 2
      O     #A316VI.StFault;	// Vibration control mill 1
      O     #A366VI.StFault;	// Vibration control mill 2
      O     #B205LS.StFault;	// Metal purifying valve closed
      O     #B206HL.StFault;	// HL DFAV full
      O     #B300SM.StFault;	// Standstill mill 1
      O     #B350SM.StFault;	// Standstill mill 2
      O     #B317HL.StFault;	// HL cone mill 1 (backup)
      O     #B367HL.StFault;	// HL cone mill 2 (backup)
      O     #Y251V_52_53_54V.StFault;	// Flap box
      O     #Ma.InAlarmTempMill1;
      O     #Ma.InAlarmTempMill2;
      AN    #Ma.InLocal;
      =     #tmpFaultStopFeedingMill2;
//--- Fault mill 1
      A     #M200.StFault;	// Fan DFAV
      O     #M300.StFault;	// Motor mill 1
      O     #DFCMMill1.StFault;	// DFCM control unit mill 1
      O     #Y203V.StFault;	// Open dense-medium valve
      O     #Y302V_Y305V.StFault;	// Cone open/close mill 1
      O     #Y307V_Y309V.StFault;	// Cone unlock/lock mill 1
      O     #A316VI.StFault;	// Vibration control mill 1
      O     #B205LS.StFault;	// Metal purifying valve closed
      O     #B206HL.StFault;	// HL DFAV full
      O     #B201LS.StFault;	// Clam-gate mill 1 closed
      O     #B300SM.StFault;	// Standstill mill 1
      O     #B310LS.StFault;	// Switch panel ok mill 1
      O     #B317HL.StFault;	// HL cone mill 1
      O     #Y251V_52_53_54V.StFault;	// Flap box
      O     #Ma.InAlarmTempMill1;
      AN    #Ma.InLocal;
      =     #Ma.OutpH311Z3;	// Alarm lamp mill 1
      =     #Ma.OutAlarmMill1;
//--- Fault mill 2
      A     #M200.StFault;	// Fan DFAV
      O     #M350.StFault;	// Motor mill 2
      O     #DFCMMill2.StFault;	// DFCM control unit mill 2
      O     #Y203V.StFault;	// Open dense-medium valve
      O     #Y352V_Y355V.StFault;	// Cone open/close mill 2
      O     #Y357V_Y359V.StFault;	// Cone unlock/lock mill 2
      O     #A366VI.StFault;	// Vibration control mill 2
      O     #B205LS.StFault;	// Metal purifying valve closed
      O     #B206HL.StFault;	// HL DFAV full
      O     #B250LS.StFault;	// Clam-gate mill 2 closed
      O     #B350SM.StFault;	// Standstill mill 2
      O     #B360LS.StFault;	// Switch panel ok mill 2
      O     #B367HL.StFault;	// HL cone mill 2
      O     #Y251V_52_53_54V.StFault;	// Flap box
      O     #Ma.InAlarmTempMill2;
      AN    #Ma.InLocal;
      A     #Ma.Par.ParWithMill2;
      =     #Ma.OutpH361Z3;	// Alarm lamp mill 2
      =     #Ma.OutAlarmMill2;
//--- Local mode --
      A     #Ma.InLocal;
      =     #M200.InLocal;
      =     #M300.InLocal;
      =     #M350.InLocal;
      =     #DFCMMill1.InLocal;
      =     #DFCMMill2.InLocal;
      =     #B205LS.InLocal;
      =     #B206HL.InLocal;
      =     #B201LS.InLocal;
      =     #B250LS.InLocal;
      =     #B300SM.InLocal;
      =     #B350SM.InLocal;
      =     #B310LS.InLocal;
      =     #B360LS.InLocal;
      =     #B317HL.InLocal;
      =     #B367HL.InLocal;
      =     #A209LC_AO1.InLocal;
      =     #A209LC_AO2.InLocal;
      =     #A209LC_AI1.InLocal;
      =     #A209LC_AI2.InLocal;
      =     #Y251V_52_53_54V.InLocal;
// Open dense-medium valve
      AN    #Ma.InpS311Z2;	// Not automatic mode mill 1
      AN    #Ma.InpS311Z2_1;	// Not service mode mill 1
      A(;
      AN    #Ma.InpS361Z2;	// Not automatic mode mill 2
      AN    #Ma.InpS361Z2_1;	// Not service mode mill 2
      ON    #Ma.Par.ParWithMill2;
      );
      =     #Y203V.InLocal;
      AN    #Ma.InUsedMill1;
      O     #Ma.InLocal;
      =     #A316VI.InLocal;
      =     #B317HL.InLocal;
      AN    #Ma.InUsedMill2;
      O     #Ma.InLocal;
      =     #A366VI.InLocal;
      =     #B367HL.InLocal;
//--- Fault Reset -------------
      A     #Ma.CmdFaultReset;
      S     #M200.CmdFaultReset;
      S     #M300.CmdFaultReset;
      S     #M350.CmdFaultReset;
      S     #DFCMMill1.CmdFaultReset;
      S     #DFCMMill2.CmdFaultReset;
      S     #Y203V.CmdFaultReset;
      S     #Y302V_Y305V.CmdFaultReset;
      S     #Y352V_Y355V.CmdFaultReset;
      S     #Y307V_Y309V.CmdFaultReset;
      S     #Y357V_Y359V.CmdFaultReset;
      S     #A316VI.CmdFaultReset;
      S     #A366VI.CmdFaultReset;
      S     #B205LS.CmdFaultReset;
      S     #B206HL.CmdFaultReset;
      S     #B201LS.CmdFaultReset;
      S     #B250LS.CmdFaultReset;
      S     #B300SM.CmdFaultReset;
      S     #B350SM.CmdFaultReset;
      S     #B310LS.CmdFaultReset;
      S     #B360LS.CmdFaultReset;
      S     #B317HL.CmdFaultReset;
      S     #B367HL.CmdFaultReset;
      S     #A209LC_AO1.CmdFaultReset;
      S     #A209LC_AO2.CmdFaultReset;
      S     #A209LC_AI1.CmdFaultReset;
      S     #A209LC_AI2.CmdFaultReset;
      S     #Y251V_52_53_54V.CmdFaultReset;
//--- Global enable mill 1---
      AN    #Ma.OutBrakeMill1;	// Brake mill 1
      AN    #Ma.Par.OutScreenChMill1;	// Screen change mill 1
      AN    #tmpFaultStopAfEmptyMill1;
      O     #Ma.OutpBrakeMill1;
      O     #Ma.OutEmptyingMill1;
      O     #Ma.Par.OutSpeedChMill1;
      A     #Ma.InEnableMill1;	// Enable mill 1
      A     #Ma.InpS311Z2;	// Automatic mode mill 1
      AN    #Ma.InpS311Z2_1;	// Not service mode mill 1
      A     #Y302V_Y305V.StLN;	// Cone closed mill 1
      A     #Y307V_Y309V.StLN;	// Cone locked mill 1
      AN    #B300SM.StFault;	// Standstill mill 1
      AN    #tmpFaultImmStopMill1;
      AN    #Ma.Par.OutSwitchChMill1;	// Change time active mill 1
      =     #tmpEnableMill1;
//--- Global enable mill 2---
      AN    #Ma.OutBrakeMill2;	// Brake mill 2
      AN    #Ma.Par.OutScreenChMill2;	// Screen change mill 2
      AN    #tmpFaultStopAfEmptyMill2;
      O     #Ma.OutpBrakeMill2;
      O     #Ma.OutEmptyingMill2;
      O     #Ma.Par.OutSpeedChMill2;
      A     #Ma.InEnableMill2;	// Enable mill 2
      A     #Ma.InpS361Z2;	// Automatic mode mill 2
      AN    #Ma.InpS361Z2_1;	// Not service mode mill 2
      A     #Y352V_Y355V.StLN;	// Cone closed mill 2
      A     #Y357V_Y359V.StLN;	// Cone locked mill 2
      AN    #B350SM.StFault;	// Standstill mill 2
      A     #Ma.Par.ParWithMill2;
      AN    #tmpFaultImmStopMill2;
      AN    #Ma.Par.OutSwitchChMill2;	// Change time active mill 2
      =     #tmpEnableMill2;
//--- Interlocking A316VI Vibration control mill 1
      SET;
      =     #A316VI.InMonTrue;
//--- Interlocking A366VI Vibration control mill 2
      SET;
      =     #A366VI.InMonTrue;
//--- Interlocking B205LS Metal purifying valve closed
      A     #Ma.OutFeedingMill1;
      O     #Ma.OutFeedingMill2;
      O     #Ma.StStarted;	// [1.3]
      =     #B205LS.InMonTrue;
//--- Interlocking B206HL HL DFAV full
      SET;
      =     #B206HL.InMonFalse;
//--- Interlocking B201LS Clam-gate mill 1 closed
      AN    #Ma.InEnableFeedMill1;
      AN    #DFCMMill1.InManual;	// [1.5]
      A     #Ma.Par.ParWithDFCM;	// [1.1]
      =     #B201LS.InMonTrue;
      AN    #Ma.Par.ParWithDFCM;	// [1.1]
      =     #B201LS.InMonFalse;	// [1.1]
//--- Interlocking B250LS Clam-gate mill 2 closed
      AN    #Ma.InEnableFeedMill2;
      AN    #DFCMMill2.InManual;	// [1.5]
      A     #Ma.Par.ParWithDFCM;	// [1.1]
      =     #B250LS.InMonTrue;
      AN    #Ma.Par.ParWithDFCM;	// [1.1]
      =     #B250LS.InMonFalse;	// [1.1]
//--- Interlocking B300SM Standstill mill 1
// Check running by enable, otherwise fault
      A     #M300.OutpRunFwd;
      O     #M300.OutpRunRev;
      =     #B300SM.InMonFalse;
//--- Interlocking B350SM Standstill mill 1
// Check running by enable, otherwise fault
      A     #M350.OutpRunFwd;
      O     #M350.OutpRunRev;
      =     #B350SM.InMonFalse;
//--- Interlocking B310LS Switch panel ok mill 1
      CLR;
      =     #B310LS.InMonTrue;
//--- Interlocking B360LS Switch panel ok mill 2
      CLR;
      =     #B360LS.InMonTrue;
//--- Interlocking B317HL HL cone mill 1
      SET;
      =     #B317HL.InMonFalse;
//--- Interlocking B367HL HL cone mill 2
      SET;
      =     #B367HL.InMonFalse;
NETWORK
TITLE = Handle speed and direction change of mill motors M300/M350
//--- Between forward <-> reverse motor must come to a standstill
      A     #B350SM.StTrue;	// Standstill mill 2
      ON    #Ma.Par.ParWithMill2;
      A     #B300SM.StTrue;	// Standstill mill 1
      A     #Ma.InOutRevMill;
      S     #Ma.OutRevMill;
      A     #B350SM.StTrue;	// Standstill mill 2
      ON    #Ma.Par.ParWithMill2;
      A     #B300SM.StTrue;	// Standstill mill 1
      AN    #Ma.InOutRevMill;
      R     #Ma.OutRevMill;
//--- Between fast to slow motor switches must be cleared
// Mill 1
      A     #Ma.InFastMill;
      AN    #Ma.OutBrakeMill1;
      A     #Ma.Par.OutSwitchChDoneMill1;
      S     #Ma.OutFastMill1;
      R     #Ma.Par.OutSwitchChDoneMill1;
      AN    #Ma.InFastMill;
      O     #Ma.OutBrakeMill1;
      A     #Ma.Par.OutSwitchChDoneMill1;
      O     #M300.StStopped;
      ON    #M300.Par.Par2Speed;
      R     #Ma.OutFastMill1;
      R     #Ma.Par.OutSwitchChDoneMill1;
// Mill 2
      A     #Ma.InFastMill;
      AN    #Ma.OutBrakeMill2;
      A     #Ma.Par.OutSwitchChDoneMill2;
      S     #Ma.OutFastMill2;
      R     #Ma.Par.OutSwitchChDoneMill2;
      AN    #Ma.InFastMill;
      O     #Ma.OutBrakeMill2;
      A     #Ma.Par.OutSwitchChDoneMill2;
      O     #M350.StStopped;
      ON    #M350.Par.Par2Speed;
      R     #Ma.OutFastMill2;
      R     #Ma.Par.OutSwitchChDoneMill2;
NETWORK
TITLE = Interlocking M300 Motor mill 1
      A(;
      AN    #Ma.OutRevMill;	// Common run forward
      AN    #Ma.OutpBrakeMill1;
      O;
      AN    #Ma.OutRevMill;	// Brake at run forward
      A     #Ma.OutpBrakeMill1;
      A     #Ma.Par.ParHwDirWhileBrake;
      O;
      A     #Ma.OutRevMill;	// Brake at run reverse
      A     #Ma.OutpBrakeMill1;
      AN    #Ma.Par.ParHwDirWhileBrake;
      );
      A     #tmpEnableMill1;
      =     #M300.InEnableFwd;	// M300 release forward
      A(;
      A     #Ma.OutRevMill;	// Common run reverse
      AN    #Ma.OutpBrakeMill1;
      O;
      A     #Ma.OutRevMill;	// Brake at run reverse
      A     #Ma.OutpBrakeMill1;
      A     #Ma.Par.ParHwDirWhileBrake;
      O;
      AN    #Ma.OutRevMill;	// Brake at run forward
      A     #Ma.OutpBrakeMill1;
      AN    #Ma.Par.ParHwDirWhileBrake;
      );
      A     #tmpEnableMill1;
      =     #M300.InEnableRev;	// M300 release forward
      AN    #Ma.OutFastMill1;
      =     #M300.InSlow;
      AN    #Ma.InBrakeMill1;
      AN    #Ma.Par.OutBrakeAcvMill1;
      O     #Ma.OutpBrakeMill1;
      O     #Ma.Par.OutSpeedChMill1;
      A     #Ma.CmdNext;
      A     #Ma.InDischargeOkMill1;	// Discharge ok mill 1
      A     #Y203V.StLN;	// Dense-medium flap closed
      AN    #B205LS.StFault;	// Metal purifying valve closed
      AN    #B206HL.StFault;	// HL DFAV full
      AN    #B201LS.StFault;	// Clam gate mill 1 not fault
      AN    #B250LS.StFault;	// Clam gate mill 2 not fault
      AN    #B317HL.StFault;	// HL cone mill 1 (backup)
      AN    #B367HL.StFault;	// HL cone mill 2 (backup)
      AN    #tmpFaultStopFeedingMill1;
      A(;	//[2.3]    
      L     #Ma.InScreenNoMill1;	//[2.3]
      L     #Ma.OutScreenNoAcMill1;	//[2.3]
      ==I;	//[2.3]
      );	//[2.3]
      S     #M300.CmdNext;
//--- Sequence stop
      A     #Ma.OutEmptyRunMill1;
      ON    #Ma.Par.ParWithDFCM;	// [0.2]
      ON    #Ma.Par.ParWithDFAV;	// [0.2]
      AN    #Ma.InEnableFeedMill1;
      A(;
      O     #M300.StStartedRev;
      O     #M300.StStartedFwd;
      );
      S     #Ma.OutEmptySeqStopMill1;
      A     #Ma.InEnableFeedMill1;
      ON    #Ma.InEnableMill1;
      ON    #Ma.InUsedMill1;
      O     #tmpSpeedChangeMill1;
      O     #Ma.OutBrakeMill1;
      R     #Ma.OutEmptySeqStopMill1;
      A     #Ma.InSeqStop;
      ON    #Ma.InUsedMill1;
      O     #Ma.OutEmptySeqStopMill1;
      AN    #Ma.OutEmptyingMill1;	// Emptying time not running
      =     #M300.InSeqStop;
NETWORK
TITLE = Interlocking M350 Motor mill 2
      A(;
      AN    #Ma.OutRevMill;	// Common run forward
      AN    #Ma.OutpBrakeMill2;
      O;
      AN    #Ma.OutRevMill;	// Brake at run forward
      A     #Ma.OutpBrakeMill2;
      A     #Ma.Par.ParHwDirWhileBrake;
      O;
      A     #Ma.OutRevMill;	// Brake at run reverse
      A     #Ma.OutpBrakeMill2;
      AN    #Ma.Par.ParHwDirWhileBrake;
      );
      A     #tmpEnableMill2;
      =     #M350.InEnableFwd;	// M350 release forward
      A(;
      A     #Ma.OutRevMill;	// Common run reverse
      AN    #Ma.OutpBrakeMill2;
      O;
      A     #Ma.OutRevMill;	// Brake at run reverse
      A     #Ma.OutpBrakeMill2;
      A     #Ma.Par.ParHwDirWhileBrake;
      O;
      AN    #Ma.OutRevMill;	// Brake at run forward
      A     #Ma.OutpBrakeMill2;
      AN    #Ma.Par.ParHwDirWhileBrake;
      );
      A     #tmpEnableMill2;
      =     #M350.InEnableRev;	// M350 release forward
      AN    #Ma.OutFastMill2;
      =     #M350.InSlow;
      AN    #Ma.InBrakeMill2;
      AN    #Ma.Par.OutBrakeAcvMill2;
      O     #Ma.OutpBrakeMill2;
      O     #Ma.Par.OutSpeedChMill2;
      A     #Ma.CmdNext;
      A     #Ma.InDischargeOkMill2;	// Discharge ok mill 2
      A     #Y203V.StLN;	// Dense-medium flap closed
      AN    #B205LS.StFault;	// Metal purifying valve closed
      AN    #B206HL.StFault;	// HL DFAV full
      AN    #B201LS.StFault;	// Clam gate mill 1 not fault
      AN    #B250LS.StFault;	// Clam gate mill 2 not fault
      AN    #B317HL.StFault;	// HL cone mill 1 (backup)
      AN    #B367HL.StFault;	// HL cone mill 2 (backup)
      AN    #tmpFaultStopFeedingMill2;
      A(;	//[2.3]    
      L     #Ma.InScreenNoMill2;	//[2.3]
      L     #Ma.OutScreenNoAcMill2;	//[2.3]
      ==I;	//[2.3]
      );	//[2.3]
      S     #M350.CmdNext;
//--- Sequence stop
      A     #Ma.OutEmptyRunMill2;
      ON    #Ma.Par.ParWithDFCM;	// [0.2]
      ON    #Ma.Par.ParWithDFAV;	// [0.2]
      AN    #Ma.InEnableFeedMill2;
      A(;
      O     #M350.StStartedRev;
      O     #M350.StStartedFwd;
      );
      S     #Ma.OutEmptySeqStopMill2;
      A     #Ma.InEnableFeedMill2;
      AN    #Ma.InSeqStop;
      A     #Ma.InUsedMill2;
      ON    #Ma.InEnableMill2;
      ON    #Ma.InUsedMill2;
      O     #tmpSpeedChangeMill2;
      O     #Ma.OutBrakeMill2;
      R     #Ma.OutEmptySeqStopMill2;
      A     #Ma.InSeqStop;
      ON    #Ma.InUsedMill2;
      O     #Ma.OutEmptySeqStopMill2;
      AN    #Ma.OutEmptyingMill2;	// Emptying time not running
      =     #M350.InSeqStop;
NETWORK
TITLE = Interlocking M200
      A     #Ma.InEnableMill1;
      O     #Ma.InEnableMill2;
      A     #Ma.Par.ParWithDFAV;
      =     #M200.InEnableFwd;
      A     #M300.StStartedFwd;
      O     #M300.StStartedRev;
      O(;
      A     #M350.StStartedFwd;
      O     #M350.StStartedRev;
      );
      A     #Ma.CmdNext;
      AN    #tmpFaultStopFeedingMill1;
      AN    #tmpFaultStopFeedingMill2;
      S     #M200.CmdNext;
      A(;	//--Case: 1 mill
      A     #B201LS.StTrue;	// Clam-gate mill 1 closed
      A     #Ma.Par.ParWithGateMill1;
      AN    #Ma.Par.ParWithMill2;
      O(;	//--Case: 2 mills, 2 gates
      A     #B201LS.StTrue;	// Clam-gate mill 1 closed
      A     #Ma.Par.ParWithGateMill1;
      A     #B250LS.StTrue;	// Clam-gate mill 2 closed
      A     #Ma.Par.ParWithGateMill2;
      A     #Ma.Par.ParWithMill2;
      );
      O(;	//--Case: 2 mills, only gate 1
      A     #B201LS.StTrue;	// Clam-gate mill 1 closed
      A     #Ma.Par.ParWithGateMill1;
      AN    #Ma.Par.ParWithGateMill2;
      A     #Ma.Par.ParWithMill2;
      );
      O(;	//--Case: 2 mills, only gate 2
      AN    #Ma.Par.ParWithGateMill1;
      A     #B250LS.StTrue;	// Clam-gate mill 2 closed
      A     #Ma.Par.ParWithGateMill2;
      A     #Ma.Par.ParWithMill2;
      );
      O(;
      A     #B201LS.StFault;	// Fault clam-gate mill 1: not closed
      O     #B250LS.StFault;	// Fault clam-gate mill 2: not closed
      );
      );
      A     #Ma.InSeqStop;
      =     #M200.InSeqStop;
NETWORK
TITLE = Interlocking DFCM Mills 1 and 2
// Programming the following functions:
// - Release DFCM (Clam-gate DFAV-1 or DFAV-2), if M200 is running
//   and DFCM is released.
      NOP   0;
//--- Feeding mill 1
      A     #Ma.Par.OutInPosFlapBox;	// Flap box in correct position
      ON    #Ma.Par.ParWithFlapBox;
      ON    #Ma.Par.ParWithMill2;
      A     #Y203V.StLN;	// Dense-medium valve is closed
      A     #B205LS.StTrue;	// Metal purifying valve closed
      A     #B206HL.StFalse;	// HL DFAV full
      A     #B317HL.StFalse;	// HL cone mill 1
      A     #tmpEnableMill1;
      AN    #tmpFaultStopFeedingMill1;
      A     #Ma.InEnableFeedMill1;
      A     #Ma.InDischargeOkMill1;
      A     #Ma.InUsedMill1;	// Mill 1 is used
      AN    #Ma.InSeqStop;
      AN    #Ma.OutBrakeMill1;
      AN    #Ma.Par.OutBrakeAcvMill1;
      AN    #tmpSpeedChangeMill1;
      A     #Ma.StStarted;
//->[1.6a] DFCM 1/2 koordinieren
      A(;
      A     #M350.StStartedFwd;
      O     #M350.StStartedRev;
      AN    #Ma.Par.OutSpeedChMill2;
      ON    #Ma.InUsedMill2;
      ON    #Ma.Par.ParWithMill2;
      );
//<-[1.6a]
      =     #DFCMMill1.InEnableFwd;
      A     #DFCMMill1.StStartedFwd;
      O;
      A     #Ma.InEnableFeedMill1;
      AN    #Ma.Par.ParWithDFAV;
      O;
      A     #Ma.InEnableFeedMill1;
      AN    #Ma.Par.ParWithDFCM;
      =     #Ma.OutFeedingMill1;
      S     #Ma.OutLoadedMill1;
      R     #Ma.OutEmptyingDoneMill1;
//--- Feeding mill 2
      A     #Ma.Par.OutInPosFlapBox;	// Flap box in correct position
      ON    #Ma.Par.ParWithFlapBox;
      A     #Y203V.StLN;	// Dense-medium valve is closed
      A     #B205LS.StTrue;	// Metal purifying valve closed
      A     #B206HL.StFalse;	// HL DFAV full
      A     #B367HL.StFalse;	// HL cone mill 2
      A     #tmpEnableMill2;
      AN    #tmpFaultStopFeedingMill2;
      A     #Ma.InEnableFeedMill2;
      A     #Ma.InDischargeOkMill2;
      A     #Ma.InUsedMill2;	// Mill 2 is used
      AN    #Ma.InSeqStop;
      AN    #Ma.OutBrakeMill2;
      AN    #Ma.Par.OutBrakeAcvMill2;
      AN    #tmpSpeedChangeMill2;
      A     #Ma.Par.ParWithMill2;
      A     #Ma.StStarted;
//->[1.6a] DFCM 1/2 koordinieren
      A(;
      A     #M300.StStartedFwd;
      O     #M300.StStartedRev;
      ON    #Ma.InUsedMill1;
      AN    #Ma.Par.OutSpeedChMill1;
      );
//<-[1.6a]
      =     #DFCMMill2.InEnableFwd;
      A     #DFCMMill2.StStartedFwd;
      O;
      A     #Ma.InEnableFeedMill2;
      AN    #Ma.Par.ParWithDFAV;
      O;
      A     #Ma.InEnableFeedMill2;
      AN    #Ma.Par.ParWithDFCM;
      =     #Ma.OutFeedingMill2;
      S     #Ma.OutLoadedMill2;
      R     #Ma.OutEmptyingDoneMill2;
//----Seq. stop / next
      CLR;
      =     #DFCMMill1.InSeqStop;
      =     #DFCMMill2.InSeqStop;
      A     #Ma.StStarted;
      S     #DFCMMill1.CmdNext;
      S     #DFCMMill2.CmdNext;
NETWORK
TITLE = Interlocking Y203V dense-medium valve
// Programming the following functions:
// - Open/close the valve to empty the dense-medium via push button
// - Control the push-button lamps S311Z5 and S361Z5. They may light on, if 
//   the dense-medium emptying is released.
//
// Lamp release for opening heavy-particle gate mill 1
//
      A(;
      A     #B201LS.StTrue;	// Clam-gate mill l closed
      A     #DFCMMill1.StStopped;	// Feeder mill 1 stopped
      A     #Ma.Par.ParWithGateMill1;
      A(;
      A     #B250LS.StTrue;	// Clam-gate mill 2 closed
      A     #DFCMMill2.StStopped;	// Feeder mill 2 stopped
      ON    #Ma.Par.ParWithGateMill2;	// [0.1]
      ON    #Ma.Par.ParWithMill2;	// [0.1]
      );
      );
      A     #Ma.Par.ParWithDFAV;
      AN    #Y203V.InLocal;
      =     #Ma.OutpS311Z5;	// Lamp release for opening heavy-particle gate mill 1
// Lamp release for opening heavy-particle gate mill 2
      A(;
      A     #B201LS.StTrue;	// Clam-gate mill l closed 
      A     #DFCMMill1.StStopped;	// Feeder mill 1 stopped
      ON    #Ma.Par.ParWithGateMill1;
      A(;
      A     #B250LS.StTrue;	// Clam-gate mill 2 closed
      A     #DFCMMill2.StStopped;	// Feeder mill 2 stopped
      A     #Ma.Par.ParWithGateMill2;	// [0.1]
      A     #Ma.Par.ParWithMill2;	// [0.1]
      );
      );
      A     #Ma.Par.ParWithDFAV;
      AN    #Y203V.InLocal;
      =     #Ma.OutpS361Z5;	// Lamp release for opening heavy-particle gate mill 2
// Dense-medium valve open/close
      A     #Ma.InpS311Z5;	// Push button open heavy-particle gate mill 1
      A     #Ma.OutpS311Z5;	// Lamp release for opening heavy-particle gate mill 1
      O;
      A     #Ma.InpS361Z5;	// Push button open heavy-particle gate mill 2
      A     #Ma.OutpS361Z5;	// Lamp release for opening heavy-particle gate mill 2
      =     #Y203V.InEnableHN;	// Open dense-medium valve
      CLR;
      =     #Y203V.InSeqStop;
      SET;
      S     #Y203V.CmdNext;
NETWORK
TITLE = Interlocking Y251V_52_53_54V Flap box
// Programming the following functions:
// - Set the flap valve-DFAV direction only mill 1, only mill 2 or both mills
// - Automatically switch to the used mills 
//
      A     #Ma.Par.ParWithMill2;
      A     #Ma.Par.ParWithFlapBox;
      JCN   eIFV;
// Set signal flap box in correct position
      A     #Ma.InUsedMill1;
      A     #Ma.InUsedMill2;
      A     #Y251V_52_53_54V.StMiddle1;	//Position mill 1 and 2
      O;
      A     #Ma.InUsedMill1;
      AN    #Ma.InUsedMill2;
      A     #Y251V_52_53_54V.StLN;	//Position mill 1
      O;
      AN    #Ma.InUsedMill1;
      A     #Ma.InUsedMill2;
      A     #Y251V_52_53_54V.StHN;	//Position mill 2
      =     #Ma.Par.OutInPosFlapBox;	// Flap box is in correct position
      A     #B201LS.StTrue;	// Clam-gate mill 1 closed
      A     #B250LS.StTrue;	// Clam-gate mill 2 closed
      A     #Ma.InUsedMill1;
      AN    #Ma.InUsedMill2;
      =     #Y251V_52_53_54V.InLN;	//Position mill 1
      A     #B201LS.StTrue;	// Clam-gate mill 1 closed
      A     #B250LS.StTrue;	// Clam-gate mill 2 closed
      AN    #Ma.InUsedMill1;
      A     #Ma.InUsedMill2;
      S     #Y251V_52_53_54V.CmdHN;	//Position mill 2
      A     #B201LS.StTrue;	// Clam-gate mill 1 closed
      A     #B250LS.StTrue;	// Clam-gate mill 2 closed
      A     #Ma.InUsedMill1;
      A     #Ma.InUsedMill2;
      S     #Y251V_52_53_54V.CmdMiddle1;	// Position mills 1 and 2
eIFV: NOP   0;
NETWORK
TITLE = Interlocking cone mill 1
// Programming the following functions:
//- Local mode
//- Open/close cone
//- Unlock/lock cone
      NOP   0;
// [0.3] Cone open/close mill 1
      A     #Ma.InpS311Z3;	// Push button open cone mill 1
      O     #Ma.InpS311Z4;	// Push button close cone mill 1
      O     #Ma.Par.OutUnlockConeMill1;	// Request unlock cone mill 1
      A     #Ma.InpS311Z2_1;	// Service mode mill 1
      A     #Y307V_Y309V.StHN;	// Cone unlocked mill 1
      O     #Ma.InpS311Z2;	// Automatic mode mill 1
      NOT;
      =     #Y302V_Y305V.InLocal;
// Cone unlock/lock mill 1
      AN    #Ma.InpS311Z2;	// Not automatic mode mill 1
      AN    #Ma.InpS311Z2_1;	// Not service mode mill 1
      A     #B300SM.InpTrue;	// Standstill mill 1
      =     #Y307V_Y309V.InLocal;
//Open cone (valve)
      A     #Ma.InpS311Z2_1;	// Service mode mill 1
      A(;
      A     #Ma.InpS311Z3;	// Push button open cone mill 1
      AN    #Ma.InpS311Z4;	// Push button close cone mill 1
      O;
      A     #Ma.InpS311Z4;	// Push button close cone mill 1
      A     #B310LS.StFalse;	// Switch panel not ok mill 1
      O;
      A     #Ma.Par.OutUnlockConeMill1;	// Request unlock cone mill 1
      );
      A     #B300SM.StTrue;	// Standstill mill 1
      A     #Y307V_Y309V.StHN;	// Cone unlocked mill 1
      AN    #Y302V_Y305V.StFault;	// Cone open/close mill 1
      AN    #Y307V_Y309V.StFault;	// Cone unlock/lock mill 1
      =     #Y302V_Y305V.InEnableHN;	// Cone open mill 1
//Lamp open cone mill 1
      AN    #Ma.InpS311Z2;	// Not automatic mode mill 1
      A     #Ma.InpS311Z2_1;	// Service mode mill 1
      A     #B300SM.StTrue;	// Standstill mill 1
      AN    #Y302V_Y305V.StFault;	// Cone open/close mill 1
      AN    #Y307V_Y309V.StFault;	// Cone unlock/lock mill 1
      AN    #Y302V_Y305V.StHN;	// Cone not opened mill 1
//[0.3]   UN      #Y302V_Y305V.InLocal;
      =     #Ma.OutpS311Z3;	// Lamp release for opening cone mill 1
//Close cone (valve)
      A     #Ma.InpS311Z2_1;	// Service mode mill 1
      A     #B300SM.StTrue;	// Standstill mill 1
      A     #Ma.InpS311Z4;	// Push button close cone mill 1
      AN    #Ma.InpS311Z3;	// Push button open cone mill 1
      A     #Y307V_Y309V.StHN;	// Cone unlocked  mill 1
      AN    #Y302V_Y305V.StLN;	// Cone not closed mill 1
      A     #B310LS.StTrue;	// Switch panel ok mill 1
      AN    #Y302V_Y305V.StFault;	// Cone open/close mill 1
      AN    #Y307V_Y309V.StFault;	// Cone unlock/lock mill 1
//[0.3]   O;
//[0.3]   UN      #Y302V_Y305V.StLN;              // Cone not closed mill 1
//[0.3]   U       #Y307V_Y309V.StLN;              // Cone locked mill 1
      =     #Y302V_Y305V.InEnableLN;	// Close cone mill 1
//Lamp close cone mill 1
      AN    #Ma.InpS311Z2;	// Not automatic mode mill 1
      A     #Ma.InpS311Z2_1;	// Service mode mill 1
      A     #B300SM.StTrue;	// Standstill mill 1
      AN    #Y302V_Y305V.StFault;	// Cone open/close mill 1
      AN    #Y307V_Y309V.StFault;	// Cone unlock/lock mill 1
      AN    #Y302V_Y305V.StLN;	// Cone not closed mill 1
      A     #B310LS.StTrue;	// Switch panel ok mill 1
//[0.3]   UN      #Y302V_Y305V.InLocal;
      =     #Ma.OutpS311Z4;	// Lamp release for closing cone mill 1
//Unlock cone (valve)
      A     #Ma.Par.OutUnlockConeMill1;	// Request unlock cone mill 1
      =     #Y307V_Y309V.InEnableHN;	// Unlock cone mill 1
//Lock cone
      A     #Y302V_Y305V.StLN;	// Cone closed mill 1
      AN    #Ma.Par.OutUnlockConeMill1;	// Request unlock cone mill 1
      A     #B310LS.StTrue;	// Switch panel ok mill 1
      =     #Y307V_Y309V.InEnableLN;	// Lock cone mill 1
//Request unlock cone (#Ma.OutUnlockConeMill1)
      AN    #Ma.InpS311Z2;	// Not automatic mode mill 1
      A     #Ma.InpS311Z2_1;	// Service mode mill 1
      A     #Ma.InpS311Z3;	// Push button open cone mill 1
      AN    #Ma.InpS311Z4;	// Push button close cone mill 1
      A     #B300SM.StTrue;	// Standstill mill 1
      A(;
      A     #Y302V_Y305V.StLN;	// Cone closed mill 1
      O     #Y302V_Y305V.StNoPosition;	// Cone closed mill 1  // [1.4]
      );
      A     #Y307V_Y309V.StLN;	// Cone locked mill 1
      AN    #Y307V_Y309V.InLocal;
      S     #Ma.Par.OutUnlockConeMill1;	// Request unlock cone mill 1
      A     #Y307V_Y309V.StHN;	// Cone unlocked mill 1
      AN    #Y302V_Y305V.InpLN;	// Cone not closed mill 1
      O     #Y302V_Y305V.StFault;	// Cone open/close mill 1
      O     #Y307V_Y309V.StFault;	// Cone unlock/lock mill 1
      R     #Ma.Par.OutUnlockConeMill1;	// Request unlock cone mill 1
      CLR;
      =     #Y302V_Y305V.InSeqStop;
      =     #Y307V_Y309V.InSeqStop;
      SET;
      S     #Y302V_Y305V.CmdNext;
      S     #Y307V_Y309V.CmdNext;
NETWORK
TITLE = Interlocking cone mill 2
// Programming the following functions:
//- Open/close cone
//- Unlock/lock cone
      NOP   0;
//[0.3] Cone open/close mill 2
      A     #Ma.InpS361Z3;	// Push button open cone mill 2
      O     #Ma.InpS361Z4;	// Push button close cone mill 2
      O     #Ma.Par.OutUnlockConeMill2;	// Request unlock cone mill 2
      A     #Ma.InpS361Z2_1;	// Service mode mill 2
      A     #Y357V_Y359V.StHN;	// Cone unlocked mill 2
      O     #Ma.InpS361Z2;	// Automatic mode mill 2
      NOT;
      =     #Y352V_Y355V.InLocal;
// Cone unlock/lock mill 2
      AN    #Ma.InpS361Z2;	// Not automatic mode mill 2
      AN    #Ma.InpS361Z2_1;	// Not service mode mill 2
      A     #B350SM.InpTrue;	// Standstill mill 2
      =     #Y357V_Y359V.InLocal;
//Open cone (valve)
      A     #Ma.InpS361Z2_1;	// Service mode mill 2
      A(;
      A     #Ma.InpS361Z3;	// Push button open cone mill 2
      AN    #Ma.InpS361Z4;	// Push button close cone mill 2
      O;
      A     #Ma.InpS361Z4;	// Push button close cone mill 2
      A     #B360LS.StFalse;	// Switch panel not ok mill 2
      O;
      A     #Ma.Par.OutUnlockConeMill2;	// Request unlock cone mill 2
      );
      A     #B350SM.StTrue;	// Standstill mill 2
      A     #Y357V_Y359V.StHN;	// Cone unlocked mill 2
      AN    #Y352V_Y355V.StFault;	// Cone open/close mill 2
      AN    #Y357V_Y359V.StFault;	// Cone unlock/lock mill 2
      =     #Y352V_Y355V.InEnableHN;	// Cone open mill 2
//Lamp open cone mill 2
      AN    #Ma.InpS361Z2;	// Not automatic mode mill 2
      A     #Ma.InpS361Z2_1;	// Service mode mill 2
      A     #B350SM.StTrue;	// Standstill mill 2
      AN    #Y352V_Y355V.StFault;	// Cone open/close mill 2
      AN    #Y357V_Y359V.StFault;	// Cone unlock/lock mill 2
      AN    #Y352V_Y355V.StHN;	// Cone not opened mill 2
//[0.3]   UN      #Y352V_Y355V.InLocal;
      =     #Ma.OutpS361Z3;	// Lamp release for opening cone mill 2
//Close cone (valve)
      A     #Ma.InpS361Z2_1;	// Service mode mill 2
      A     #B350SM.StTrue;	// Standstill mill 2
      A     #Ma.InpS361Z4;	// Push button close cone mill 2
      AN    #Ma.InpS361Z3;	// Push button open cone mill 2
      A     #Y357V_Y359V.StHN;	// Cone unlocked  mill 2
      AN    #Y352V_Y355V.StLN;	// Cone not closed mill 2
      A     #B360LS.StTrue;	// Switch panel ok mill 2
      AN    #Y352V_Y355V.StFault;	// Cone open/close mill 2
      AN    #Y357V_Y359V.StFault;	// Cone unlock/lock mill 2
//[0.3]   O;
//[0.3]   UN      #Y352V_Y355V.StLN;              // Cone not closed mill 2
//[0.3]   U       #Y357V_Y359V.StLN;              // Cone locked mill 2
      =     #Y352V_Y355V.InEnableLN;	// Close cone mill 2
//Lamp close cone mill 2
      AN    #Ma.InpS361Z2;	// Not automatic mode mill 2
      A     #Ma.InpS361Z2_1;	// Service mode mill 2
      A     #B350SM.StTrue;	// Standstill mill 2
      AN    #Y352V_Y355V.StFault;	// Cone open/close mill 2
      AN    #Y357V_Y359V.StFault;	// Cone unlock/lock mill 2
      AN    #Y352V_Y355V.StLN;	// Cone not closed mill 2
      A     #B360LS.StTrue;	// Switch panel ok mill 2
//[0.3]   UN      #Y352V_Y355V.InLocal;
      =     #Ma.OutpS361Z4;	// Lamp release for closing cone mill 2
//Unlock cone (valve)
      A     #Ma.Par.OutUnlockConeMill2;	// Request unlock cone mill 2
      =     #Y357V_Y359V.InEnableHN;	// Unlock cone mill 2
//Lock cone
      A     #Y352V_Y355V.StLN;	// Cone closed mill 2
      AN    #Ma.Par.OutUnlockConeMill2;	// Request unlock cone mill 2
      A     #B360LS.StTrue;	// Switch panel ok mill 2
      =     #Y357V_Y359V.InEnableLN;	// Lock cone mill 2
//Request unlock cone (#Ma.OutUnlockConeMill2)
      AN    #Ma.InpS361Z2;	// Not automatic mode mill 2
      A     #Ma.InpS361Z2_1;	// Service mode mill 2
      A     #Ma.InpS361Z3;	// Push button open cone mill 2
      AN    #Ma.InpS361Z4;	// Push button close cone mill 2
      A     #B350SM.StTrue;	// Standstill mill 2
      A(;
      A     #Y352V_Y355V.StLN;	// Cone closed mill 2
      O     #Y352V_Y355V.StNoPosition;	// Cone closed mill 2  // [1.4]
      );
      A     #Y357V_Y359V.StLN;	// Cone locked mill 2
      AN    #Y357V_Y359V.InLocal;
      S     #Ma.Par.OutUnlockConeMill2;	// Request unlock cone mill 2
      A     #Y357V_Y359V.StHN;	// Cone unlocked mill 2
      AN    #Y352V_Y355V.InpLN;	// Cone not closed mill 2
      O     #Y352V_Y355V.StFault;	// Cone open/close mill 2
      O     #Y357V_Y359V.StFault;	// Cone unlock/lock mill 2
      R     #Ma.Par.OutUnlockConeMill2;	// Request unlock cone mill 2
      CLR;
      =     #Y352V_Y355V.InSeqStop;
      =     #Y357V_Y359V.InSeqStop;
      SET;
      S     #Y352V_Y355V.CmdNext;
      S     #Y357V_Y359V.CmdNext;
NETWORK
TITLE = Call motor: M200 Fan DFAV
      A     #Ma.Par.ParWithDFAV;
      JCN   el2;
      CALL  #M200;
NETWORK
TITLE = Call motor: M300 Motor mill 1
// Simulate inputs if braking motor mill 2
el2:  A     #M300.InpRunFwd;
      O     #Ma.OutpBrakeMill1;
      A     #M300.OutpRunFwd;
      =     #M300.InpRunFwd;
      A     #M300.InpRunRev;
      O     #Ma.OutpBrakeMill1;
      A     #M300.OutpRunRev;
      =     #M300.InpRunRev;
      A     #M300.InpRunSlow;
      O     #Ma.OutpBrakeMill1;
      A     #M300.OutpRunSlow;
      =     #M300.InpRunSlow;
      A     #M300.InpRunFast;
      O     #Ma.OutpBrakeMill1;
      A     #M300.OutpRunFast;
      =     #M300.InpRunFast;
      CALL  #M300;
NETWORK
TITLE = Call motor: M350 Motor mill 2
      A     #Ma.Par.ParWithMill2;
      JCN   el4;
// Simulate inputs if braking motor mill 2
      A     #M350.InpRunFwd;
      O     #Ma.OutpBrakeMill2;
      A     #M350.OutpRunFwd;
      =     #M350.InpRunFwd;
      A     #M350.InpRunRev;
      O     #Ma.OutpBrakeMill2;
      A     #M350.OutpRunRev;
      =     #M350.InpRunRev;
      A     #M350.InpRunSlow;
      O     #Ma.OutpBrakeMill2;
      A     #M350.OutpRunSlow;
      =     #M350.InpRunSlow;
      A     #M350.InpRunFast;
      O     #Ma.OutpBrakeMill2;
      A     #M350.OutpRunFast;
      =     #M350.InpRunFast;
// call element
      CALL  #M350;
NETWORK
TITLE = Call motor: DFCMMill1 DFCM control unit mill 1
el4:  A     #Ma.Par.ParWithDFAV;
      A     #Ma.Par.ParWithDFCM;
      JCN   el5;
      CALL  #DFCMMill1;
NETWORK
TITLE = Call motor: DFCMMill2 DFCM control unit mill 2
el5:  A     #Ma.Par.ParWithMill2;
      A     #Ma.Par.ParWithDFAV;
      A     #Ma.Par.ParWithDFCM;
      JCN   el6;
      CALL  #DFCMMill2;
NETWORK
TITLE = Call VLS: Y203V Open dense-medium valve
el6:  A     #Ma.Par.ParWithDFAV;
      JCN   el7;
      CALL  #Y203V;
// [1.1] Enable open flap in fault state
      A     #Y203V.OutpHN;
      O;
      A     #Y203V.StFault;
      A     #Y203V.InEnableHN;
      =     #Y203V.OutpHN;
NETWORK
TITLE = Call VLS: Y302V_Y305V Cone open/close mill 1
el7:  CALL  #Y302V_Y305V;
NETWORK
TITLE = Call VLS: Y352V_Y355V Cone open/close mill 2
      A     #Ma.Par.ParWithMill2;
      JCN   el9;
      CALL  #Y352V_Y355V;
NETWORK
TITLE = Call VLS: Y307V_Y309V Cone unlock/lock mill 1
el9:  CALL  #Y307V_Y309V;
NETWORK
TITLE = Call VLS: Y357V_Y359V Cone unlock/lock mill 2
      A     #Ma.Par.ParWithMill2;
      JCN   el11;
      CALL  #Y357V_Y359V;
NETWORK
TITLE = Call Digital Input: A316VI Vibration control mill 1
el11: CALL  #A316VI;
NETWORK
TITLE = Call Digital Input: A366VI Vibration control mill 1
      A     #Ma.Par.ParWithMill2;
      JCN   el13;
      CALL  #A366VI;
NETWORK
TITLE = Call Digital Input: B205LS Metal purifying valve closed
el13: A     #Ma.Par.ParWithDFAV;
      JCN   el14;
      CALL  #B205LS;
NETWORK
TITLE = Call Digital Input: B206HL HL DFAV full
el14: A     #Ma.Par.ParWithDFAV;
      JCN   el15;
      CALL  #B206HL;
NETWORK
TITLE = Call Digital Input: B201LS Clam-gate mill 1 closed
el15: A     #Ma.Par.ParWithGateMill1;
      A     #Ma.Par.ParWithDFAV;
// [1.1]     U    #Ma.Par.ParWithDFCM;
      JCN   el16;
      CALL  #B201LS;
NETWORK
TITLE = Call Digital Input: B250LS Clam-gate mill 2 closed
el16: A     #Ma.Par.ParWithMill2;
      A     #Ma.Par.ParWithGateMill2;
      A     #Ma.Par.ParWithDFAV;
// [1.1]  U       #Ma.Par.ParWithDFCM;
      JCN   el17;
      CALL  #B250LS;
NETWORK
TITLE = Call Digital Input: B300SM Standstill mill 1
el17: CALL  #B300SM;
NETWORK
TITLE = Call Digital Input: B350SM Standstill mill 2
      A     #Ma.Par.ParWithMill2;
      JCN   el19;
      CALL  #B350SM;
NETWORK
TITLE = Call Digital Input: B310LS Switch panel ok mill 1
el19: CALL  #B310LS;
NETWORK
TITLE = Call Digital Input: B360LS Switch panel ok mill 2
      A     #Ma.Par.ParWithMill2;
      JCN   el21;
      CALL  #B360LS;
NETWORK
TITLE = Call Digital Input: B317HL HL cone mill 1
el21: CALL  #B317HL;
NETWORK
TITLE = Call Digital Input: B367HL HL cone mill 2
      A     #Ma.Par.ParWithMill2;
      JCN   el23;
      CALL  #B367HL;
NETWORK
TITLE = Call Analog Output: A209LC_AO1 Setpoint mill 1
el23: A     #Ma.Par.ParWithDFAV;
      A     #Ma.Par.ParWithDFCM;
      JCN   el24;
      CALL  #A209LC_AO1;
NETWORK
TITLE = Call Analog Output: A209LC_AO2 Setpoint mill 2
el24: A     #Ma.Par.ParWithMill2;
      A     #Ma.Par.ParWithDFAV;
      A     #Ma.Par.ParWithDFCM;
      JCN   el25;
      CALL  #A209LC_AO2;
NETWORK
TITLE = Call Analog Input: A209LC_AI1 Actual value mill 1
// A209LC_AI1: Actual load motor mill 1 [0.01 %]
el25: A     #Ma.Par.ParWithDFAV;
      A     #Ma.Par.ParWithDFCM;
      JCN   el26;
      CALL  #A209LC_AI1;
      L     #A209LC_AI1.OutValuePc;	// Actual load [0.01 %]
      L     #Ma.Par.ParEmptyRunMill1;
      <=I;
      =     #Ma.OutEmptyRunMill1;
NETWORK
TITLE = Call Analog Input: A209LC_AI2 Actual value mill 2
// A209LC_AI2: Actual load motor mill 2 [0.01 %]
el26: A     #Ma.Par.ParWithMill2;
      A     #Ma.Par.ParWithDFAV;
      A     #Ma.Par.ParWithDFCM;
      JCN   el27;
      CALL  #A209LC_AI2;
      L     #A209LC_AI2.OutValuePc;	// Actual load [0.01 %]
      L     #Ma.Par.ParEmptyRunMill2;
      <=I;
      =     #Ma.OutEmptyRunMill2;
NETWORK
TITLE = Call VLS4: Y251V_52_53_54V Flap box
el27: A     #Ma.Par.ParWithMill2;
      A     #Ma.Par.ParWithFlapBox;
      JCN   el28;
      CALL  #Y251V_52_53_54V;
el28: NOP   0;
NETWORK
TITLE = Transition to StStarting
      A(;
      A     #M350.StStarting;
      A     #Ma.Par.ParWithMill2;
      O;
      A     #M200.StStarting;
      A     #Ma.Par.ParWithDFAV;
      O     #M300.StStarting;
      );
      A(;
      O     #Ma.StStopped;
      O     #Ma.StStarted;
      O     #Ma.StStopping;
      );
      R     #Ma.StStopped;
      R     #Ma.StStarted;
      R     #Ma.StStopping;
      S     #Ma.StStarting;
NETWORK
TITLE = Transition to StStarted
      A     #M300.StStartedFwd;
      O     #M300.StStartedRev;
      ON    #Ma.InUsedMill1;
      AN    #Ma.Par.OutSpeedChMill1;	//[1.6a] Mill1 statt Mill2
      A(;
      A     #M350.StStartedFwd;
      O     #M350.StStartedRev;
      AN    #Ma.Par.OutSpeedChMill2;
      ON    #Ma.InUsedMill2;
      ON    #Ma.Par.ParWithMill2;
      );
      A(;
      A     #M200.StStartedFwd;
      ON    #Ma.Par.ParWithDFAV;
      A(;	// ParWithDFAV=0: one of the mill motors must run
      O     #M300.StStartedFwd;
      O     #M300.StStartedRev;
      O     #M350.StStartedFwd;
      O     #M350.StStartedRev;
      );
      );
      A(;
      O     #Ma.StStopped;
      O     #Ma.StStarting;
      O     #Ma.StStopping;
      );
      R     #Ma.StStopped;
      R     #Ma.StStarting;
      R     #Ma.StStopping;
      S     #Ma.StStarted;
NETWORK
TITLE = Transition to StStopping
      A(;
      A     #M350.StStopping;
      A     #Ma.Par.ParWithMill2;
      A     #Ma.InUsedMill2;	// [1.6]
      O;
      A     #M300.StStopping;
      A     #Ma.InUsedMill1;	// [1.6]
      O;
      A     #M200.StStopping;
      A     #Ma.Par.ParWithDFAV;
      );
      A(;
      O     #Ma.StStarted;
      O     #Ma.StStarting;
      );
      O     #Ma.StFault;
      AN    #tmpFaultSum;
      R     #Ma.StStarted;
      R     #Ma.StStarting;
      R     #Ma.StFault;
      S     #Ma.StStopping;
// Transition StStarted -> StStopping
      A(;
      AN    #M300.StStartedFwd;
      AN    #M300.StStartedRev;
      A     #Ma.InUsedMill1;
      O;
      AN    #M350.StStartedFwd;
      AN    #M350.StStartedRev;
      A     #Ma.Par.ParWithMill2;
      A     #Ma.InUsedMill2;
      O;
      AN    #M200.StStartedFwd;
      A     #Ma.Par.ParWithDFAV;
      O;	// [1.6]
      AN    #Ma.InUsedMill1;	// [1.6]
      AN    #Ma.InUsedMill2;	// [1.6]
      );
      A     #Ma.StStarted;
      R     #Ma.StStarted;
      S     #Ma.StStopping;
NETWORK
TITLE = Transition to StStopped
      A(;
      A     #M300.StStopped;
      A     #B300SM.StTrue;	// Standstill mill 1
      A(;
      A     #M350.StStopped;
      A     #B350SM.StTrue;	// Standstill mill 2
      ON    #Ma.Par.ParWithMill2;
      );
      A(;
      A     #M200.StStopped;
      ON    #Ma.Par.ParWithDFAV;
      );
      A(;
      A     #B201LS.StTrue;	// Clam-gate mill 1 closed
      ON    #Ma.Par.ParWithGateMill1;
      ON    #Ma.Par.ParWithDFAV;
      ON    #Ma.Par.ParWithDFCM;
      );
      A(;
      A     #B250LS.StTrue;	// Clam-gate mill 2 closed
      ON    #Ma.Par.ParWithMill2;
      ON    #Ma.Par.ParWithGateMill1;
      ON    #Ma.Par.ParWithDFAV;
      ON    #Ma.Par.ParWithDFCM;
      );
      );
      A     #Ma.StStopping;
      O;
      AN    #Ma.StStopped;	// Initialise state
      AN    #Ma.StStarting;
      AN    #Ma.StStarted;
      AN    #Ma.StStopping;
      AN    #Ma.StFault;
      R     #Ma.StStopping;
      =     #tmpTriggerFlag;
      S     #Ma.StStopped;
      A     #tmpTriggerFlag;
      AN    #Ma.InOutRevMill;	//--Change direction of mill motors:
      S     #Ma.InOutRevMill;	// Motor will be started reverse at next start
      JC    S0ed;
      A     #tmpTriggerFlag;
      A     #Ma.InOutRevMill;
      R     #Ma.InOutRevMill;	// Motor will be started forward at next start
S0ed: NOP   0;
NETWORK
TITLE = Transition to StFault
      A     #tmpFaultSum;
      R     #Ma.StStopped;
      R     #Ma.StStarting;
      R     #Ma.StStarted;
      R     #Ma.StStopping;
      S     #Ma.StFault;
NETWORK
TITLE = State Code
// State                 StCode
// -----------------------------
// StFault                 32
// StStopped                1
// StStarting               2
// StStarted.Wait           3
// StStarted.Feeding        4
// StStopping               7
// StWarning                8
      A     #Ma.StStopped;
      L     1;	//Code=StStopped
      JC    Code;
      O     #Ma.OutFeedingMill1;
      O     #Ma.OutFeedingMill2;
      A     #Ma.StStarted;
      L     4;	// Code= StStarted.Feeding
      JC    Code;
      A     #Ma.StStarted;
      L     3;	// Code=StStarted.Wait
      JC    Code;
      A     #Ma.StStarting;
      L     2;	//Code=StStarting
      JC    Code;
      A     #Ma.StStopping;
      L     7;	//Code=StStopping 
      JC    Code;
      L     32;	//Code=StFault 
Code: L     #Ma.StCode;	// Old state code
      TAK;
      T     #Ma.StCode;	// Save state code
      <>I;
      L     3;
      CC    "SYS_CBitCtrl";	//Set change bit
NETWORK
TITLE = Global End
      SET;	//---Clear all commands
      R     #Ma.CmdNext;
      R     #Ma.CmdFaultReset;
      R     #Ma.CmdTick100ms;
NETWORK
TITLE = Init Manual mode when not in Automatic mode 
      NOP   0;
//[2.2]--->
      AN    #Ma.InpS311Z2;	// not Automatic mode mill 1
      A     #M300.InManual;
      R     #M300.InManual;
      R     #M300.OutpRunFwd;
      R     #M300.OutpRunRev;
      R     #M300.OutpRunSlow;
      R     #M300.OutpRunFast;
      AN    #Ma.InpS361Z2;	// not Automatic mode mill 2
      A     #M350.InManual;
      R     #M350.InManual;
      R     #M350.OutpRunFwd;
      R     #M350.OutpRunRev;
      R     #M350.OutpRunSlow;
      R     #M350.OutpRunFast;
//<--[2.2]
END_FUNCTION_BLOCK

FUNCTION_BLOCK "GCS7_M_Discharger"	// FB 56
TITLE = Bin discharger A
//COPYRIGHT:    (C) 1997  BUHLER AG, CH-9240 UZWIL, SWITZERLAND
//
//PRODUCT:      GCS7
//
//TITLE:        FB 56 Machine Control:Bin discharger A 
//              VLS or motor, vibro , LL and Flow
//
//-------------------------------------------------------------------------
//
//IDENT:        AUTHOR:             DEPT:                       DATE:
//
//FB56.4.4      A. Egli             BASE                        25-Mar-2008
//              - Flowmonitor functionallity also without Bin-LL
//FB56.4.3      A. Egli             CT3                         13-Feb-2008
//              Vibro: Interlock CmdNext with Ma.CmdNext
//FB56.4.2      A. Egli             CT3                         22-Jun-2004
//              Test Ma.Par.ParVibroOnTime <>0
//FB56.4.1      A. Egli             CT3                         12-Sep-2003
//              Vibro.CmdNext only when vibro is enabled 
//FB56.4.0      A. Egli             CT3                         17-Jun-2002
//              New Release with one block 
//              Fast pulsing if Flow is uncovered an LL is covered
//              Flowmonitor handling corrected (3.7)
//FB56.3.5      A. Egli             CT3                         29-Oct-2001
//              LL.InLocal moved to last segment
//FB56.3.4      A. Egli             CT3                         04-Jan-2001
//              Handling of flowmonitor corrected without vibro
//FB56.3.3      Ph. Engler          MU664                       07-Dec-2000
//              Handling of flowmonitor corrected
//FB56.3.2      A. Egli             CT3                         26-Jan-2000
//              BinEmpty
//FB56.3.1      A. Egli             CT3                         21-Jan-2000
//              CmdNext of Discharger adapted
//FB56.3.0      A. Egli             CT3                         11-Oct-1999
//              Local data reduced 
//FB56.2C       A. Egli             CT3                         26-Apr-1999
//              Check ParWithVibro
//FB56.2B       K. Tischer          MU664                       06-Mrz-1999
//              CC FC2 not UC FC2
//FB56.2C       A. Egli             CT3                         20-Oct-1998
//              InDisableVibro
//FB56.2A       A. Egli             CT3                         04-Mai-1998
//              StFault = StCode 32
//FB56.1A       A.Egli              AEE61                       05-Jul-1997
//              1st Release in S7
//
//-------------------------------------------------------------------------
//
//PURPOSE:      MANUAL : see [LL.DSAxxMAN]
//
//RESTRICTIONS: S7
//              ACCU2: Pointer to dynamic datas of the machine
//              ACCU1: Pointer to parameter datas of the machine
//
//-------------------------------------------------------------------------
//
//
AUTHOR : EA
FAMILY : GCS7LL
NAME : Discharg
VERSION : 4.4
VAR
  Ma : UDT 20560;
  Discharger : FB 12;	//Element for VLS(FB13) or Motor(FB12)
  Vibro : FB 12;	//Element
  Flow : FB 14;	//Element
END_VAR
VAR_TEMP
  tmpFaultStop : BOOL ;
  tmpFaultSum : BOOL ;
  tmpNext : BOOL ;
  tmpLenDyn : INT ;
  tmpStoreAR2 : DINT ;
END_VAR
BEGIN
NETWORK
TITLE =
      L     22;
      T     #tmpLenDyn;
NETWORK
TITLE = PC Control
//=== Test Object number =====================
      L     "SYS_DirectCtrlDB".PC.ObjectNo;	//PCControl.ObjectNo
      L     #Ma.Par.ParObjectNo;	//Input ObjectNo
      <>I;
      JC    aEnd;
//=== Test OType      ========================
      L     2056;	//Input object type
      L     "SYS_DirectCtrlDB".PC.ObjectType;	//PCControl.ObjectType
      <>I;
      JC    aEnd;
//=== Test Handshake =========================
      A     "SYS_DirectCtrlDB".PC.Hsk.FExamine;	// Handshake.FExamine
      JC    aExa;
      A     "SYS_DirectCtrlDB".PC.Hsk.FDefineCmd;	// Handshake.FDefineCmd
      JC    aCmd;
      A     "SYS_DirectCtrlDB".PC.Hsk.FDefinePara;	// Handshake.FDefinePara
      JC    aPar;
aIni: L     2;	// FcInit
      UC    "SYS_DirectCtrl";
      JU    aEnd;
// Write parameter 
aPar: LAR1  P#DBX 58.0;
      L     P#6.0;
      +AR1;
      L     DBW [AR1,P#4.0];
      T     #Ma.Par.ParVibroOnTime;
      L     DBW [AR1,P#6.0];
      T     #Ma.Par.ParVibroOffTime;
      L     DBW [AR1,P#8.0];
      T     #Ma.Par.ParRestDischargeTime;
// Write new commands from PC to Interface of group 
aCmd: A     "SYS_DirectCtrlDB".PC.Cmd1[8];	//Cmd1[8]=CmdOff
      S     #Ma.CmdOff;
      A     "SYS_DirectCtrlDB".PC.Cmd1[9];	//Cmd1[9]=CmdOn
      S     #Ma.CmdOn;
      A     "SYS_DirectCtrlDB".PC.Cmd1[10];	//Cmd1[10]=CmdNext
      S     #Ma.CmdNext;
      A     "SYS_DirectCtrlDB".PC.Cmd1[11];	//Cmd1[11]=CmdFaultReset
      S     #Ma.CmdFaultReset;
      A     "SYS_DirectCtrlDB".PC.Cmd1[13];	//Cmd1[13]=CmdManualOn
      S     #Ma.InManual;
      A     "SYS_DirectCtrlDB".PC.Cmd1[6];	//Cmd1[6]=SlowOn
      A     #Ma.Par.ParDischargerIsMotor;
      S     #Discharger.InOutManSlow;
      A     "SYS_DirectCtrlDB".PC.Cmd2[6];	//Cmd2[6]=SlowOff
      A     #Ma.Par.ParDischargerIsMotor;
      R     #Discharger.InOutManSlow;
      A     "SYS_DirectCtrlDB".PC.Cmd1[1];	//Cmd1[1]=CmdRestDischargeOn
      S     #Ma.InRestDischarge;
      A     "SYS_DirectCtrlDB".PC.Cmd2[1];	//Cmd2[1]=CmdRestDischargeOff
      R     #Ma.InRestDischarge;
      A     "SYS_DirectCtrlDB".PC.Cmd1[2];	//Cmd1[1]=CmdDisableVibroOn
      S     #Ma.InDisableVibro;
      A     "SYS_DirectCtrlDB".PC.Cmd2[2];	//Cmd2[1]=CmdDisableVibroOff
      R     #Ma.InDisableVibro;
      JU    aIni;
aExa: TAR2;	// Address Dynamic data
      T     "SYS_DirectCtrlDB".GC.InDynAddr;	// -->PCControl.GC.InDynAddr
      L     #tmpLenDyn;	// Length Dynamic data
      T     "SYS_DirectCtrlDB".GC.InDynLen;	// -->PCControl.GC.InDynLen
      L     0;
      T     "SYS_DirectCtrlDB".GC.InParaAddr;	// -->PCControl.GC.InParaAddr
      T     "SYS_DirectCtrlDB".GC.InParaLen;	// -->PCControl.GC.InParaLen
      L     1;	// Code FcExamine
      UC    "SYS_DirectCtrl";
      L     10;	//Revision
      T     "SYS_DirectCtrlDB".GC.Revision;
aEnd: NOP   0;
NETWORK
TITLE = Interlocking
//===Global Group Orders===
      A     "GCS7_Gr_OutManualOn";	//Gr.OutManualOn
      S     #Ma.InManual;
      A     "GCS7_Gr_OutManualOff";	//Gr.OutManualOff
      R     #Ma.InManual;
      A     #Ma.InManual;
      S     "GCS7_Gr_InManual";	//Gr.InManual
      A     #Ma.CmdNext;
      AN    #Ma.InManual;
      O     #Ma.CmdOn;
      =     #tmpNext;
//---- Low level 
      A     #Ma.InUncovered;	//[4.0]
      ON    #Ma.Par.ParWithLL;
      A(;
      A     #Flow.StFalse;	//[3.2]
      O     #Flow.StCtoTrue;	//[3.2]
      O     #Flow.StFault;	//[3.2]
      ON    #Ma.Par.ParWithFlow;	//[3.2]
      );
      =     #Ma.OutUncovered;
      A     #Ma.OutRestDischarged;
      A     #Ma.OutUncovered;
      O;
      A     #Ma.OutUncovered;
      AN    #Ma.InRestDischarge;
      =     #Ma.OutEmpty;
//--- Fault----
      A     #Flow.StFault;
      O     #Discharger.StFault;
      O     #Vibro.StFault;
      =     #tmpFaultSum;
// 
//--- Interlocking Discharger 
      A     #Ma.InEnable;
      A     #tmpNext;
      S     #Discharger.InEnableFwd;	//Discharger.InEnableHN; 
      AN    #Ma.InEnable;
      O     #Ma.CmdOff;
      R     #Discharger.InEnableFwd;	//Discharger.InEnableHN; 
      A     #Ma.Par.ParDischargerIsMotor;
      JC    inJ1;
      AN    #Discharger.InEnableFwd;	//Discharger.InEnableHN; 
      =     #Discharger.InEnableRev;	//=Discharger.InEnableLN 
      S     #Discharger.CmdNext;
      JU    inJ2;
inJ1: CLR;
      =     #Discharger.InEnableRev;
inJ2: A     #tmpNext;	// 3.1:
      S     #Discharger.CmdNext;	// 3.1:
// 
//--- Interlocking Vibro
//      U     #Ma.Par.ParWithFlow         //[3.6]
//      UN    #Flow.StTrue                //[3.6]
//      U(                                //[3.6]
//      U     #Ma.InCovered               //[3.6]
//      U     #Ma.Par.ParWithLL           //[3.6]
//      )     
      O     #Ma.OutPulseVibroOn;
      O     #Ma.Par.ParContinuous;
      A     #Discharger.InEnableFwd;	//Discharger.InEnableHN; 
      A     #Discharger.StStartedFwd;	//Discharger.StHN; 
      AN    #Ma.InDisableVibro;
      AN    #Flow.StFault;
      =     #Vibro.InEnableFwd;
      A     #Vibro.InEnableFwd;	//[4.1]
      A     #tmpNext;	//[4.3]
      S     #Vibro.CmdNext;
// 
//--- Monitoring Flow
      A     #Discharger.StStartedFwd;	//Discharger.StHN; 
      O     #Flow.StFalse;	//[3.7]
      A(;	//[3.7]
      A     #Ma.InCovered;	//[3.7]  [4.0]
      ON    #Ma.Par.ParWithLL;	//[3.7]
      );	//[3.7]
      AN    #Flow.StFault;	//[3.7]
      =     #Flow.InMonTrue;	//[3.7]
      A(;	//[3.7]
      O     #Discharger.StStopped;	//[3.7]
      O     #Discharger.StStarting;	//[3.7]
      );	//[3.7]
      AN    #Flow.StTrue;	//[3.7]
      AN    #Flow.StCtoFalse;	//[3.7]
      S     #Flow.CmdRunTimeoutTime;	//[3.7]
// 
//--- Local mode --
      A     #Ma.InLocal;
      AN    #Ma.InManual;
      =     #Vibro.InLocal;
      =     #Flow.InLocal;
      A     #Ma.Par.ParDischargerIsMotor;
      ON    #Discharger.StStopped;	//Discharger.StLN;
      A     #Ma.InLocal;
      AN    #Ma.InManual;
      =     #Discharger.InLocal;
//--- Fault Reset -------------
      A     #Ma.CmdFaultReset;
      S     #Discharger.CmdFaultReset;
      S     #Vibro.CmdFaultReset;
      S     #Flow.CmdFaultReset;
//== Timer rest discharge
      A     #Ma.OutUncovered;
      JC    T1J1;
      R     #Ma.OutRestDischarged;
      L     0;
      T     #Ma.Par.OutRestDischargeTime;
      JU    T1J2;
T1J1: AN    "GCS7_Gr_OutTick200ms";	//Gr.OutTick200ms
      ON    #Ma.StStarted;
      O     #Ma.OutRestDischarged;
      JC    T1J2;
      L     #Ma.Par.OutRestDischargeTime;
      +     2;
      T     #Ma.Par.OutRestDischargeTime;
      L     #Ma.Par.ParRestDischargeTime;
      >I;
      S     #Ma.OutRestDischarged;
T1J2: NOP   0;
NETWORK
TITLE = Call Discharger
      A     #Ma.Par.ParDischargerIsMotor;
      JC    D_M;
      TAR2  #tmpStoreAR2;
      L     P##Discharger;
      L     DW#16#FFFFFF;
      AD;
      +AR2;
      UC    "GCS7_E_ValveControl";	//VLS FB13
      LAR2  #tmpStoreAR2;
      JU    DVLS;
D_M:  CALL  #Discharger;
DVLS: NOP   0;
NETWORK
TITLE = Call Vibro
      AN    #Ma.Par.ParWithVibro;
      JC    el4;
      CALL  #Vibro;
NETWORK
TITLE = Call Digital Input: Flow
el4:  AN    #Ma.Par.ParWithFlow;
      JC    StJ0;
      CALL  #Flow;
NETWORK
TITLE = Jump to actual state
StJ0: A     #Ma.StStopped;
      JC    S0;	// ===> State
      A     #Ma.StStarted;
      JC    S2;	// ===> State
      A     #Ma.StStarting;
      JC    S1;	// ===> State
      A     #Ma.StStopping;
      JC    S3;	// ===> State
      A     #Ma.StFault;
      JC    S4;	// ===> State
NETWORK
TITLE = Stopped
//any Transition 
xxS0: S     #Ma.StStopped;	// ===> Initialisation
      JU    OUT;
//=== Logic
// Condition for StFault
S0:   A     #tmpFaultSum;
      R     #Ma.StStopped;
      JC    xxS4;	//--> ST_FAULT:
// Condition for StStarting
      AN    #Vibro.StStopped;
      A     #Ma.Par.ParWithVibro;
      ON    #Discharger.StStopped;	//Discharger.StLN;
      R     #Ma.StStopped;
      JC    xxS1;	//--> StStarting
      JU    OUT;
NETWORK
TITLE = StStarting
//any Transition 
xxS1: S     #Ma.StStarting;
      JU    OUT;
//=== Logic
// Condition for StFault
S1:   A     #tmpFaultSum;
      R     #Ma.StStarting;
      JC    xxS4;	//--> StFault
// Condition for StStarted
      A     #Discharger.StStartedFwd;	//Discharger.StHN; 
      R     #Ma.StStarting;
      JC    xxS2;	//-->StStarted
// Condition for StStopping
      AN    #Discharger.StStarting;	//Discharger.StCtoHN;
      R     #Ma.StStarting;
      JC    xxS3;	//-->StStopping
      JU    OUT;
NETWORK
TITLE = StStarted
//any Transition 
xxS2: S     #Ma.StStarted;
      S     #Ma.OutPulseVibroOn;
      L     0;
      T     #Ma.Par.OutDelayTime;
      T     #Ma.Par.OutRestDischargeTime;
      JU    OUT;
//=== Logic
// Condition for StFault
S2:   A     #tmpFaultSum;
      R     #Ma.StStarted;
      JC    xxS4;	//--> StFault
// Condition for StStopping
      AN    #Discharger.StStartedFwd;	//Discharger.StHN;
      R     #Ma.StStarted;
      JC    xxS3;	//-->StStopping
//== timer Vibro
//Start Vibro immediatly at negativ flag of
      A     #Ma.InCovered;	//[3.6]
      ON    #Ma.Par.ParWithLL;	//[3.6] [4.4]
      A     #Ma.Par.ParWithFlow;	//[3.6]
      A     #Flow.StTrue;	//[3.6]
      FN    #Ma.OutEdgeFlowCovered;	//[3.6]
      JCN   S2J1;	//[3.6]
      L     0;	//[3.6]
      T     #Ma.Par.OutDelayTime;	//[3.6]
      S     #Ma.OutPulseVibroOn;	//[3.6]
S2J1: AN    "GCS7_Gr_OutTick200ms";	//Gr.OutTick200ms
      JC    OUT;
      L     #Ma.Par.OutDelayTime;
      +     2;
      T     #Ma.Par.OutDelayTime;
      A     #Ma.OutPulseVibroOn;
      JC    S2On;
//Vibro off time
      A     #Ma.InCovered;	//[3.6]
      ON    #Ma.Par.ParWithLL;	//[3.6] [4.4]
      A     #Ma.Par.ParWithFlow;	//[3.6]
      AN    #Flow.StTrue;	//[3.6]
      L     #Ma.Par.ParVibroOnTime;	//[3.6]
      SRW   1;	//[3.6]
      JC    S2F2;	//[3.6]
      L     #Ma.Par.ParVibroOffTime;
S2F2: L     #Ma.Par.OutDelayTime;
      >=I;
      JC    OUT;
      S     #Ma.OutPulseVibroOn;
      JU    S2J0;
//Vibro on time
S2On: L     #Ma.Par.ParVibroOnTime;
      <I;
      JC    OUT;
      R     #Ma.OutPulseVibroOn;
S2J0: L     0;
      T     #Ma.Par.OutDelayTime;
      JU    OUT;
NETWORK
TITLE = Stopping
//any Transition 
xxS3: S     #Ma.StStopping;
      R     #Ma.OutPulseVibroOn;
      JU    OUT;
//=== Logic
// Condition for StFault
S3:   A     #tmpFaultSum;
      R     #Ma.StStopping;
      JC    xxS4;	//--> StFault
// Condition for StStopped
      A     #Vibro.StStopped;
      ON    #Ma.Par.ParWithVibro;
      A     #Discharger.StStopped;	//Discharger.StLN; 
      R     #Ma.StStopping;
      JC    xxS0;	//-->StStopped
// Condition for StStarting
      AN    #Discharger.StStopping;	//Discharger.StCtoLN;
      AN    #Discharger.StStopped;	//Discharger.StLN;
      R     #Ma.StStopping;
      JC    xxS1;	//-->StStarting
      JU    OUT;
NETWORK
TITLE = Fault
//any Transition 
xxS4: S     #Ma.StFault;
      JU    OUT;
//=== Logic
S4:   A     #tmpFaultSum;
      JC    OUT;
//---- Transition --
      R     #Ma.StFault;
      JU    xxS0;	//-->StStopping 
NETWORK
TITLE = State Code
// State     StCode
// ----------------------
// StFault32
// StStopped    1
// StStarting   2
// StStarted    3
// StStopping  7
OUT:  A     #Ma.StStopped;
      L     1;	//Code=StStopped
      JC    Code;
      AN    #Discharger.OutpRunSlow;
      A     #Ma.Par.ParDischargerIsMotor;
      A     #Ma.StStarted;
      L     3;	//Code=StStartedSlow
      JC    Code;
      A     #Ma.StStarted;
      L     4;	//Code=StStartedFast
      JC    Code;
      A     #Ma.StStarting;
      L     2;	//Code=StStarting
      JC    Code;
      A     #Ma.StStopping;
      L     7;	//Code=StStopping 
      JC    Code;
      L     32;	//Code=StFault 
Code: L     #Ma.StCode;	// Old state code
      TAK;
      T     #Ma.StCode;	// Save state code
      <>I;
      L     3;
      CC    "SYS_CBitCtrl";	//Set change bit
NETWORK
TITLE = Global End
      CLR;	//---Clear all commands
      =     #Ma.CmdOn;
      =     #Ma.CmdOff;
      =     #Ma.CmdNext;
      =     #Ma.CmdFaultReset;
      L     #Ma.Par.ParVibroOnTime;	//[4.2]
      L     0;	//[4.2]
      ==I;	//[4.2]
      R     #Ma.OutPulseVibroOn;	//[4.2]
END_FUNCTION_BLOCK

